LIN {X 0,Y 401.03,Z 373.683,A -85,B 0,C 180,E1 -11453.633,E2 -11453.633} C_VEL
LIN {X 0,Y 401.846,Z 358.726,A -85,B 0,C 180,E1 -11454.448,E2 -11454.448} C_VEL
LIN {X 0,Y 397.42,Z 344.712,A -85,B 0,C 180,E1 -11455.362,E2 -11455.362} C_VEL
LIN {X 0,Y 391.491,Z 329.461,A -85,B 0,C 180,E1 -11456.225,E2 -11456.225} C_VEL
LIN {X 0,Y 390.297,Z 326.311,A -85,B 0,C 180,E1 -11456.415,E2 -11456.415} C_VEL
LIN {X 0,Y 390.293,Z 322.173,A -85,B 0,C 180,E1 -11459.09,E2 -11459.09} C_VEL
LIN {X 0,Y 390.321,Z 317.773,A -85,B 0,C 180,E1 -11462.192,E2 -11462.192} C_VEL
LIN {X 0,Y 390.35,Z 313.687,A -85,B 0,C 180,E1 -11465.179,E2 -11465.179} C_VEL
LIN {X 0,Y 390.43,Z 310.287,A -85,B 0,C 180,E1 -11467.736,E2 -11467.736} C_VEL
LIN {X 0,Y 390.446,Z 306.037,A -85,B 0,C 180,E1 -11470.887,E2 -11470.887} C_VEL
LIN {X 0,Y 390.052,Z 302.527,A -85,B 0,C 180,E1 -11473.545,E2 -11473.545} C_VEL
LIN {X 0,Y 390.057,Z 302.527,A -85,B 0,C 180,E1 -11476.789,E2 -11476.789} C_VEL
LIN {X 0,Y 390.056,Z 302.524,A -85,B 0,C 180,E1 -11479.56,E2 -11479.56} C_VEL
LIN {X 0,Y 390.042,Z 302.525,A -85,B 0,C 180,E1 -11482.449,E2 -11482.449} C_VEL
LIN {X 0,Y 390.068,Z 302.518,A -85,B 0,C 180,E1 -11485.975,E2 -11485.975} C_VEL
LIN {X 0,Y 390.036,Z 302.519,A -85,B 0,C 180,E1 -11489.7,E2 -11489.7} C_VEL
LIN {X 0,Y 390.033,Z 302.52,A -85,B 0,C 180,E1 -11493.226,E2 -11493.226} C_VEL
LIN {X 0,Y 390.069,Z 302.521,A -85,B 0,C 180,E1 -11496.763,E2 -11496.763} C_VEL
LIN {X 0,Y 390.103,Z 302.515,A -85,B 0,C 180,E1 -11499.983,E2 -11499.983} C_VEL
LIN {X 0,Y 390.138,Z 302.5,A -85,B 0,C 180,E1 -11503.248,E2 -11503.248} C_VEL
LIN {X 0,Y 390.195,Z 302.506,A -85,B 0,C 180,E1 -11506.561,E2 -11506.561} C_VEL
LIN {X 0,Y 390.167,Z 302.502,A -85,B 0,C 180,E1 -11509.623,E2 -11509.623} C_VEL
LIN {X 0,Y 390.247,Z 302.493,A -85,B 0,C 180,E1 -11512.758,E2 -11512.758} C_VEL
LIN {X 0,Y 390.211,Z 302.492,A -85,B 0,C 180,E1 -11514.833,E2 -11514.833} C_VEL
LIN {X 0,Y 390.418,Z 302.476,A -85,B 0,C 180,E1 -11517.937,E2 -11517.937} C_VEL
LIN {X 0,Y 390.549,Z 302.445,A -85,B 0,C 180,E1 -11520,E2 -11520} C_VEL
LIN {X 0,Y 390.273,Z 302.496,A -85,B 0,C 180,E1 -11523.097,E2 -11523.097} C_VEL
LIN {X 0,Y 390.301,Z 302.482,A -85,B 0,C 180,E1 -11526.202,E2 -11526.202} C_VEL
LIN {X 0,Y 390.194,Z 302.502,A -85,B 0,C 180,E1 -11529.329,E2 -11529.329} C_VEL
LIN {X 0,Y 390.171,Z 302.506,A -85,B 0,C 180,E1 -11532.483,E2 -11532.483} C_VEL
LIN {X 0,Y 390.138,Z 302.501,A -85,B 0,C 180,E1 -11535.677,E2 -11535.677} C_VEL
LIN {X 0,Y 390.102,Z 302.519,A -85,B 0,C 180,E1 -11538.922,E2 -11538.922} C_VEL
LIN {X 0,Y 390.036,Z 302.515,A -85,B 0,C 180,E1 -11542.234,E2 -11542.234} C_VEL
LIN {X 0,Y 390.049,Z 302.516,A -85,B 0,C 180,E1 -11545.722,E2 -11545.722} C_VEL
LIN {X 0,Y 390.032,Z 302.526,A -85,B 0,C 180,E1 -11549.112,E2 -11549.112} C_VEL
LIN {X 0,Y 390.042,Z 302.524,A -85,B 0,C 180,E1 -11552.721,E2 -11552.721} C_VEL
LIN {X 0,Y 390.055,Z 302.523,A -85,B 0,C 180,E1 -11555.825,E2 -11555.825} C_VEL
LIN {X 0,Y 390.065,Z 302.523,A -85,B 0,C 180,E1 -11559.218,E2 -11559.218} C_VEL
LIN {X 0,Y 390.042,Z 302.546,A -85,B 0,C 180,E1 -11561.744,E2 -11561.744} C_VEL
LIN {X 0,Y 392.326,Z 311.892,A -85,B 0,C 180,E1 -11565.039,E2 -11565.039} C_VEL
LIN {X 0,Y 395.159,Z 323.516,A -85,B 0,C 180,E1 -11568.849,E2 -11568.849} C_VEL
LIN {X 0,Y 398.138,Z 335.816,A -85,B 0,C 180,E1 -11572.593,E2 -11572.593} C_VEL
LIN {X 0,Y 398.472,Z 338.892,A -85,B 0,C 180,E1 -11573.469,E2 -11573.469} C_VEL
LIN {X 0,Y 396.461,Z 351.383,A -85,B 0,C 180,E1 -11576.665,E2 -11576.665} C_VEL
LIN {X 0,Y 394.575,Z 365.042,A -85,B 0,C 180,E1 -11580.085,E2 -11580.085} C_VEL
LIN {X 0,Y 392.745,Z 380.859,A -85,B 0,C 180,E1 -11583.952,E2 -11583.952} C_VEL
LIN {X 0,Y 396.794,Z 403.736,A -85,B 0,C 180,E1 -11584.777,E2 -11584.777} C_VEL
LIN {X 0,Y 398.586,Z 417.426,A -85,B 0,C 180,E1 -11585.407,E2 -11585.407} C_VEL
LIN {X 0,Y 399.347,Z 429.472,A -85,B 0,C 180,E1 -11586.051,E2 -11586.051} C_VEL
LIN {X 0,Y 398.063,Z 444.07,A -85,B 0,C 180,E1 -11586.911,E2 -11586.911} C_VEL
LIN {X 0,Y 396.506,Z 458.695,A -85,B 0,C 180,E1 -11588.011,E2 -11588.011} C_VEL
LIN {X 0,Y 394.957,Z 472.268,A -85,B 0,C 180,E1 -11589.289,E2 -11589.289} C_VEL
LIN {X 0,Y 393.553,Z 484.615,A -85,B 0,C 180,E1 -11590.709,E2 -11590.709} C_VEL
LIN {X 0,Y 392.203,Z 495.885,A -85,B 0,C 180,E1 -11592.264,E2 -11592.264} C_VEL
LIN {X 0,Y 391.183,Z 505.396,A -85,B 0,C 180,E1 -11593.831,E2 -11593.831} C_VEL
LIN {X 0,Y 390.271,Z 514.747,A -85,B 0,C 180,E1 -11595.664,E2 -11595.664} C_VEL
LIN {X 0,Y 389.615,Z 522.521,A -85,B 0,C 180,E1 -11597.499,E2 -11597.499} C_VEL
LIN {X 0,Y 389.166,Z 529.796,A -85,B 0,C 180,E1 -11599.596,E2 -11599.596} C_VEL
LIN {X 0,Y 389.001,Z 535.531,A -85,B 0,C 180,E1 -11601.69,E2 -11601.69} C_VEL
LIN {X 0,Y 389.046,Z 539.872,A -85,B 0,C 180,E1 -11603.778,E2 -11603.778} C_VEL
LIN {X 0,Y 389.039,Z 542.91,A -85,B 0,C 180,E1 -11605.856,E2 -11605.856} C_VEL
LIN {X 0,Y 389.189,Z 544.737,A -85,B 0,C 180,E1 -11607.93,E2 -11607.93} C_VEL
LIN {X 0,Y 389.08,Z 545.347,A -85,B 0,C 180,E1 -11610,E2 -11610} C_VEL
LIN {X 0,Y 389.187,Z 544.737,A -85,B 0,C 180,E1 -11612.07,E2 -11612.07} C_VEL
LIN {X 0,Y 389.089,Z 542.914,A -85,B 0,C 180,E1 -11614.144,E2 -11614.144} C_VEL
LIN {X 0,Y 389.076,Z 539.867,A -85,B 0,C 180,E1 -11616.222,E2 -11616.222} C_VEL
LIN {X 0,Y 389.06,Z 535.519,A -85,B 0,C 180,E1 -11618.309,E2 -11618.309} C_VEL
LIN {X 0,Y 389.195,Z 529.78,A -85,B 0,C 180,E1 -11620.404,E2 -11620.404} C_VEL
LIN {X 0,Y 389.64,Z 522.506,A -85,B 0,C 180,E1 -11622.501,E2 -11622.501} C_VEL
LIN {X 0,Y 390.283,Z 514.721,A -85,B 0,C 180,E1 -11624.336,E2 -11624.336} C_VEL
LIN {X 0,Y 391.158,Z 505.355,A -85,B 0,C 180,E1 -11626.17,E2 -11626.17} C_VEL
LIN {X 0,Y 392.253,Z 495.847,A -85,B 0,C 180,E1 -11627.734,E2 -11627.734} C_VEL
LIN {X 0,Y 393.271,Z 486.53,A -85,B 0,C 180,E1 -11629.035,E2 -11629.035} C_VEL
LIN {X 0,Y 394.675,Z 474.561,A -85,B 0,C 180,E1 -11630.455,E2 -11630.455} C_VEL
LIN {X 0,Y 396.187,Z 461.487,A -85,B 0,C 180,E1 -11631.735,E2 -11631.735} C_VEL
LIN {X 0,Y 397.585,Z 448.807,A -85,B 0,C 180,E1 -11632.748,E2 -11632.748} C_VEL
LIN {X 0,Y 398.922,Z 434.386,A -85,B 0,C 180,E1 -11633.673,E2 -11633.673} C_VEL
LIN {X 0,Y 399.351,Z 427.194,A -85,B 0,C 180,E1 -11634.06,E2 -11634.06} C_VEL
LIN {X 0,Y 398.169,Z 411.419,A -85,B 0,C 180,E1 -11634.857,E2 -11634.857} C_VEL
LIN {X 0,Y 397.083,Z 401.601,A -85,B 0,C 180,E1 -11635.344,E2 -11635.344} C_VEL
LIN {X 0,Y 394.918,Z 387.953,A -85,B 0,C 180,E1 -11636.086,E2 -11636.086} C_VEL
LIN {X 0,Y 392.929,Z 378.662,A -85,B 0,C 180,E1 -11636.619,E2 -11636.619} C_VEL
LIN {X 0,Y 394.825,Z 365.115,A -85,B 0,C 180,E1 -11640.19,E2 -11640.19} C_VEL
LIN {X 0,Y 396.932,Z 354.413,A -85,B 0,C 180,E1 -11643.291,E2 -11643.291} C_VEL
LIN {X 0,Y 399.879,Z 343.943,A -85,B 0,C 180,E1 -11646.696,E2 -11646.696} C_VEL
LIN {X 0,Y 399.578,Z 340.879,A -85,B 0,C 180,E1 -11647.996,E2 -11647.996} C_VEL
LIN {X 0,Y 398.234,Z 335.574,A -85,B 0,C 180,E1 -11650.767,E2 -11650.767} C_VEL
LIN {X 0,Y 397.006,Z 331.283,A -85,B 0,C 180,E1 -11653.662,E2 -11653.662} C_VEL
LIN {X 0,Y 395.994,Z 328.116,A -85,B 0,C 180,E1 -11656.691,E2 -11656.691} C_VEL
LIN {X 0,Y 395.412,Z 326.545,A -85,B 0,C 180,E1 -11658.881,E2 -11658.881} C_VEL
LIN {X 0,Y 394.819,Z 325.339,A -85,B 0,C 180,E1 -11661.557,E2 -11661.557} C_VEL
LIN {X 0,Y 394.321,Z 324.865,A -85,B 0,C 180,E1 -11663.974,E2 -11663.974} C_VEL
LIN {X 0,Y 393.477,Z 325.038,A -85,B 0,C 180,E1 -11667.599,E2 -11667.599} C_VEL
LIN {X 0,Y 392.817,Z 325.946,A -85,B 0,C 180,E1 -11671.244,E2 -11671.244} C_VEL
LIN {X 0,Y 392.385,Z 327.254,A -85,B 0,C 180,E1 -11674.541,E2 -11674.541} C_VEL
LIN {X 0,Y 392.066,Z 328.943,A -85,B 0,C 180,E1 -11677.887,E2 -11677.887} C_VEL
LIN {X 0,Y 391.986,Z 329.43,A -85,B 0,C 180,E1 -11678.684,E2 -11678.684} C_VEL
LIN {X 0,Y 393.349,Z 332.348,A -85,B 0,C 180,E1 -11678.997,E2 -11678.997} C_VEL
LIN {X 0,Y 398.107,Z 342.204,A -85,B 0,C 180,E1 -11680.134,E2 -11680.134} C_VEL
LIN {X 0,Y 401.264,Z 350.393,A -85,B 0,C 180,E1 -11681.049,E2 -11681.049} C_VEL
LIN {X 0,Y 400.997,Z 355.665,A -85,B 0,C 180,E1 -11681.457,E2 -11681.457} C_VEL
LIN {X 0,Y 399.708,Z 367.932,A -85,B 0,C 180,E1 -11682.503,E2 -11682.503} C_VEL
LIN {X 0,Y 398.232,Z 379.64,A -85,B 0,C 180,E1 -11683.73,E2 -11683.73} C_VEL
LIN {X 0,Y 396.864,Z 390.351,A -85,B 0,C 180,E1 -11685.121,E2 -11685.121} C_VEL
LIN {X 0,Y 395.58,Z 399.819,A -85,B 0,C 180,E1 -11686.646,E2 -11686.646} C_VEL
LIN {X 0,Y 394.376,Z 407.68,A -85,B 0,C 180,E1 -11688.174,E2 -11688.174} C_VEL
LIN {X 0,Y 393.313,Z 414.086,A -85,B 0,C 180,E1 -11689.707,E2 -11689.707} C_VEL
LIN {X 0,Y 392.54,Z 419.208,A -85,B 0,C 180,E1 -11691.247,E2 -11691.247} C_VEL
LIN {X 0,Y 391.71,Z 423.284,A -85,B 0,C 180,E1 -11692.785,E2 -11692.785} C_VEL
LIN {X 0,Y 391.315,Z 425.442,A -85,B 0,C 180,E1 -11693.814,E2 -11693.814} C_VEL
LIN {X 0,Y 390.95,Z 428.372,A -85,B 0,C 180,E1 -11695.877,E2 -11695.877} C_VEL
LIN {X 0,Y 390.674,Z 429.276,A -85,B 0,C 180,E1 -11696.906,E2 -11696.906} C_VEL
LIN {X 0,Y 390.434,Z 429.786,A -85,B 0,C 180,E1 -11697.937,E2 -11697.937} C_VEL
LIN {X 0,Y 390.308,Z 429.858,A -85,B 0,C 180,E1 -11698.968,E2 -11698.968} C_VEL
LIN {X 0,Y 390.151,Z 428.837,A -85,B 0,C 180,E1 -11701.032,E2 -11701.032} C_VEL
LIN {X 0,Y 390.034,Z 427.759,A -85,B 0,C 180,E1 -11702.065,E2 -11702.065} C_VEL
LIN {X 0,Y 389.964,Z 426.237,A -85,B 0,C 180,E1 -11703.099,E2 -11703.099} C_VEL
LIN {X 0,Y 390.195,Z 423.138,A -85,B 0,C 180,E1 -11704.649,E2 -11704.649} C_VEL
LIN {X 0,Y 390.507,Z 419.028,A -85,B 0,C 180,E1 -11706.199,E2 -11706.199} C_VEL
LIN {X 0,Y 390.863,Z 412.829,A -85,B 0,C 180,E1 -11708.01,E2 -11708.01} C_VEL
LIN {X 0,Y 391.364,Z 404.933,A -85,B 0,C 180,E1 -11709.823,E2 -11709.823} C_VEL
LIN {X 0,Y 391.878,Z 396.479,A -85,B 0,C 180,E1 -11711.378,E2 -11711.378} C_VEL
LIN {X 0,Y 392.607,Z 386.139,A -85,B 0,C 180,E1 -11712.93,E2 -11712.93} C_VEL
LIN {X 0,Y 393.342,Z 375.598,A -85,B 0,C 180,E1 -11714.222,E2 -11714.222} C_VEL
LIN {X 0,Y 394.133,Z 362.595,A -85,B 0,C 180,E1 -11715.514,E2 -11715.514} C_VEL
LIN {X 0,Y 394.779,Z 351.319,A -85,B 0,C 180,E1 -11716.416,E2 -11716.416} C_VEL
LIN {X 0,Y 395.172,Z 338.606,A -85,B 0,C 180,E1 -11717.231,E2 -11717.231} C_VEL
LIN {X 0,Y 391.437,Z 324.013,A -85,B 0,C 180,E1 -11718.105,E2 -11718.105} C_VEL
LIN {X 0,Y 389.442,Z 316.377,A -85,B 0,C 180,E1 -11718.495,E2 -11718.495} C_VEL
LIN {X 0,Y 389.452,Z 313.434,A -85,B 0,C 180,E1 -11721.157,E2 -11721.157} C_VEL
LIN {X 0,Y 389.474,Z 309.821,A -85,B 0,C 180,E1 -11724.521,E2 -11724.521} C_VEL
LIN {X 0,Y 389.487,Z 306.163,A -85,B 0,C 180,E1 -11727.979,E2 -11727.979} C_VEL
LIN {X 0,Y 389.532,Z 303.708,A -85,B 0,C 180,E1 -11730.343,E2 -11730.343} C_VEL
LIN {X 0,Y 389.562,Z 302.588,A -85,B 0,C 180,E1 -11731.546,E2 -11731.546} C_VEL
LIN {X 0,Y 389.926,Z 302.541,A -85,B 0,C 180,E1 -11735.224,E2 -11735.224} C_VEL
LIN {X 0,Y 390.041,Z 302.524,A -85,B 0,C 180,E1 -11737.78,E2 -11737.78} C_VEL
LIN {X 0,Y 390.059,Z 302.52,A -85,B 0,C 180,E1 -11740.821,E2 -11740.821} C_VEL
LIN {X 0,Y 390.057,Z 302.519,A -85,B 0,C 180,E1 -11743.886,E2 -11743.886} C_VEL
LIN {X 0,Y 390.065,Z 302.573,A -85,B 0,C 180,E1 -11746.623,E2 -11746.623} C_VEL
LIN {X 0,Y 390.479,Z 305.87,A -85,B 0,C 180,E1 -11749.107,E2 -11749.107} C_VEL
LIN {X 0,Y 390.433,Z 310.221,A -85,B 0,C 180,E1 -11752.375,E2 -11752.375} C_VEL
LIN {X 0,Y 390.33,Z 315.186,A -85,B 0,C 180,E1 -11756.071,E2 -11756.071} C_VEL
LIN {X 0,Y 390.32,Z 320.392,A -85,B 0,C 180,E1 -11759.8,E2 -11759.8} C_VEL
LIN {X 0,Y 390.263,Z 325.586,A -85,B 0,C 180,E1 -11763.243,E2 -11763.243} C_VEL
LIN {X 0,Y 390.271,Z 326.34,A -85,B 0,C 180,E1 -11763.717,E2 -11763.717} C_VEL
LIN {X 0,Y 394.457,Z 336.878,A -85,B 0,C 180,E1 -11764.277,E2 -11764.277} C_VEL
LIN {X 0,Y 399.267,Z 350.24,A -85,B 0,C 180,E1 -11765.087,E2 -11765.087} C_VEL
LIN {X 0,Y 401.888,Z 359.314,A -85,B 0,C 180,E1 -11765.683,E2 -11765.683} C_VEL
LIN {X 0,Y 400.935,Z 374.28,A -85,B 0,C 180,E1 -11766.497,E2 -11766.497} C_VEL
LIN {X 0,Y 399.752,Z 388.734,A -85,B 0,C 180,E1 -11767.518,E2 -11767.518} C_VEL
LIN {X 0,Y 398.42,Z 401.781,A -85,B 0,C 180,E1 -11768.665,E2 -11768.665} C_VEL
LIN {X 0,Y 397.026,Z 413.662,A -85,B 0,C 180,E1 -11769.933,E2 -11769.933} C_VEL
LIN {X 0,Y 395.681,Z 424.75,A -85,B 0,C 180,E1 -11771.354,E2 -11771.354} C_VEL
LIN {X 0,Y 394.294,Z 434.875,A -85,B 0,C 180,E1 -11772.896,E2 -11772.896} C_VEL
LIN {X 0,Y 392.9,Z 444.714,A -85,B 0,C 180,E1 -11774.691,E2 -11774.691} C_VEL
LIN {X 0,Y 391.888,Z 452.947,A -85,B 0,C 180,E1 -11776.518,E2 -11776.518} C_VEL
LIN {X 0,Y 390.902,Z 460.609,A -85,B 0,C 180,E1 -11778.593,E2 -11778.593} C_VEL
LIN {X 0,Y 390.19,Z 466.693,A -85,B 0,C 180,E1 -11780.671,E2 -11780.671} C_VEL
LIN {X 0,Y 389.699,Z 471.393,A -85,B 0,C 180,E1 -11782.747,E2 -11782.747} C_VEL
LIN {X 0,Y 389.383,Z 474.836,A -85,B 0,C 180,E1 -11784.822,E2 -11784.822} C_VEL
LIN {X 0,Y 389.298,Z 477.097,A -85,B 0,C 180,E1 -11786.895,E2 -11786.895} C_VEL
LIN {X 0,Y 389.012,Z 478.268,A -85,B 0,C 180,E1 -11788.965,E2 -11788.965} C_VEL
LIN {X 0,Y 389.012,Z 478.282,A -85,B 0,C 180,E1 -11791.035,E2 -11791.035} C_VEL
LIN {X 0,Y 389.279,Z 477.166,A -85,B 0,C 180,E1 -11793.105,E2 -11793.105} C_VEL
LIN {X 0,Y 389.382,Z 474.962,A -85,B 0,C 180,E1 -11795.178,E2 -11795.178} C_VEL
LIN {X 0,Y 389.704,Z 471.482,A -85,B 0,C 180,E1 -11797.305,E2 -11797.305} C_VEL
LIN {X 0,Y 390.147,Z 466.955,A -85,B 0,C 180,E1 -11799.33,E2 -11799.33} C_VEL
LIN {X 0,Y 390.91,Z 460.581,A -85,B 0,C 180,E1 -11801.511,E2 -11801.511} C_VEL
LIN {X 0,Y 391.87,Z 453.34,A -85,B 0,C 180,E1 -11803.482,E2 -11803.482} C_VEL
LIN {X 0,Y 392.934,Z 444.959,A -85,B 0,C 180,E1 -11805.354,E2 -11805.354} C_VEL
LIN {X 0,Y 392.757,Z 441.59,A -85,B 0,C 180,E1 -11806.057,E2 -11806.057} C_VEL
LIN {X 0,Y 390.887,Z 435.993,A -85,B 0,C 180,E1 -11807.228,E2 -11807.228} C_VEL
LIN {X 0,Y 389.054,Z 430.043,A -85,B 0,C 180,E1 -11808.36,E2 -11808.36} C_VEL
LIN {X 0,Y 388.921,Z 425.982,A -85,B 0,C 180,E1 -11808.99,E2 -11808.99} C_VEL
LIN {X 0,Y 390.227,Z 414.843,A -85,B 0,C 180,E1 -11810.463,E2 -11810.463} C_VEL
LIN {X 0,Y 391.894,Z 402.013,A -85,B 0,C 180,E1 -11811.846,E2 -11811.846} C_VEL
LIN {X 0,Y 393.303,Z 388.866,A -85,B 0,C 180,E1 -11813.01,E2 -11813.01} C_VEL
LIN {X 0,Y 394.564,Z 374.255,A -85,B 0,C 180,E1 -11814.045,E2 -11814.045} C_VEL
LIN {X 0,Y 395.332,Z 360.445,A -85,B 0,C 180,E1 -11814.821,E2 -11814.821} C_VEL
LIN {X 0,Y 390.892,Z 346.436,A -85,B 0,C 180,E1 -11815.774,E2 -11815.774} C_VEL
LIN {X 0,Y 385.604,Z 332.648,A -85,B 0,C 180,E1 -11816.593,E2 -11816.593} C_VEL
LIN {X 0,Y 383.337,Z 326.923,A -85,B 0,C 180,E1 -11816.914,E2 -11816.914} C_VEL
LIN {X 0,Y 383.334,Z 322.682,A -85,B 0,C 180,E1 -11819.671,E2 -11819.671} C_VEL
LIN {X 0,Y 383.344,Z 317.471,A -85,B 0,C 180,E1 -11823.367,E2 -11823.367} C_VEL
LIN {X 0,Y 383.37,Z 313.6,A -85,B 0,C 180,E1 -11826.233,E2 -11826.233} C_VEL
LIN {X 0,Y 383.496,Z 309.036,A -85,B 0,C 180,E1 -11829.673,E2 -11829.673} C_VEL
LIN {X 0,Y 383.438,Z 306.884,A -85,B 0,C 180,E1 -11831.287,E2 -11831.287} C_VEL
LIN {X 0,Y 383,Z 303.406,A -85,B 0,C 180,E1 -11834.023,E2 -11834.023} C_VEL
LIN {X 0,Y 383.01,Z 303.404,A -85,B 0,C 180,E1 -11837.24,E2 -11837.24} C_VEL
LIN {X 0,Y 383.013,Z 303.398,A -85,B 0,C 180,E1 -11840.414,E2 -11840.414} C_VEL
LIN {X 0,Y 383.025,Z 303.397,A -85,B 0,C 180,E1 -11844.044,E2 -11844.044} C_VEL
LIN {X 0,Y 382.987,Z 303.404,A -85,B 0,C 180,E1 -11847.578,E2 -11847.578} C_VEL
LIN {X 0,Y 382.976,Z 303.398,A -85,B 0,C 180,E1 -11850.299,E2 -11850.299} C_VEL
LIN {X 0,Y 383.002,Z 303.392,A -85,B 0,C 180,E1 -11854.045,E2 -11854.045} C_VEL
LIN {X 0,Y 382.993,Z 303.396,A -85,B 0,C 180,E1 -11857.334,E2 -11857.334} C_VEL
LIN {X 0,Y 383.058,Z 303.395,A -85,B 0,C 180,E1 -11860.716,E2 -11860.716} C_VEL
LIN {X 0,Y 383.081,Z 303.383,A -85,B 0,C 180,E1 -11864.027,E2 -11864.027} C_VEL
LIN {X 0,Y 383.136,Z 303.376,A -85,B 0,C 180,E1 -11867.284,E2 -11867.284} C_VEL
LIN {X 0,Y 383.143,Z 303.385,A -85,B 0,C 180,E1 -11870.498,E2 -11870.498} C_VEL
LIN {X 0,Y 383.241,Z 303.356,A -85,B 0,C 180,E1 -11873.683,E2 -11873.683} C_VEL
LIN {X 0,Y 383.385,Z 303.352,A -85,B 0,C 180,E1 -11877.899,E2 -11877.899} C_VEL
LIN {X 0,Y 383.518,Z 303.321,A -85,B 0,C 180,E1 -11880,E2 -11880} C_VEL
LIN {X 0,Y 383.211,Z 303.376,A -85,B 0,C 180,E1 -11883.154,E2 -11883.154} C_VEL
LIN {X 0,Y 383.259,Z 303.359,A -85,B 0,C 180,E1 -11886.317,E2 -11886.317} C_VEL
LIN {X 0,Y 383.144,Z 303.38,A -85,B 0,C 180,E1 -11889.502,E2 -11889.502} C_VEL
LIN {X 0,Y 383.125,Z 303.388,A -85,B 0,C 180,E1 -11893.536,E2 -11893.536} C_VEL
LIN {X 0,Y 383.094,Z 303.382,A -85,B 0,C 180,E1 -11897.454,E2 -11897.454} C_VEL
LIN {X 0,Y 383.028,Z 303.39,A -85,B 0,C 180,E1 -11900.647,E2 -11900.647} C_VEL
LIN {X 0,Y 383.013,Z 303.403,A -85,B 0,C 180,E1 -11903.809,E2 -11903.809} C_VEL
LIN {X 0,Y 382.991,Z 303.394,A -85,B 0,C 180,E1 -11907.307,E2 -11907.307} C_VEL
LIN {X 0,Y 382.981,Z 303.404,A -85,B 0,C 180,E1 -11910.919,E2 -11910.919} C_VEL
LIN {X 0,Y 383.017,Z 303.399,A -85,B 0,C 180,E1 -11914.668,E2 -11914.668} C_VEL
LIN {X 0,Y 382.996,Z 303.404,A -85,B 0,C 180,E1 -11917.903,E2 -11917.903} C_VEL
LIN {X 0,Y 383.014,Z 303.55,A -85,B 0,C 180,E1 -11921.209,E2 -11921.209} C_VEL
LIN {X 0,Y 385.349,Z 313.104,A -85,B 0,C 180,E1 -11924.661,E2 -11924.661} C_VEL
LIN {X 0,Y 387.987,Z 324.048,A -85,B 0,C 180,E1 -11928.348,E2 -11928.348} C_VEL
LIN {X 0,Y 390.441,Z 334.196,A -85,B 0,C 180,E1 -11931.536,E2 -11931.536} C_VEL
LIN {X 0,Y 391.584,Z 339.187,A -85,B 0,C 180,E1 -11933.041,E2 -11933.041} C_VEL
LIN {X 0,Y 390.582,Z 345.973,A -85,B 0,C 180,E1 -11934.845,E2 -11934.845} C_VEL
LIN {X 0,Y 388.287,Z 360.674,A -85,B 0,C 180,E1 -11938.643,E2 -11938.643} C_VEL
LIN {X 0,Y 386.353,Z 375.405,A -85,B 0,C 180,E1 -11942.364,E2 -11942.364} C_VEL
LIN {X 0,Y 385.859,Z 379.755,A -85,B 0,C 180,E1 -11943.448,E2 -11943.448} C_VEL
LIN {X 0,Y 389.905,Z 402.276,A -85,B 0,C 180,E1 -11944.271,E2 -11944.271} C_VEL
LIN {X 0,Y 391.981,Z 417.492,A -85,B 0,C 180,E1 -11944.993,E2 -11944.993} C_VEL
LIN {X 0,Y 392.739,Z 430.161,A -85,B 0,C 180,E1 -11945.696,E2 -11945.696} C_VEL
LIN {X 0,Y 391.357,Z 444.834,A -85,B 0,C 180,E1 -11946.594,E2 -11946.594} C_VEL
LIN {X 0,Y 389.847,Z 458.096,A -85,B 0,C 180,E1 -11947.615,E2 -11947.615} C_VEL
LIN {X 0,Y 388.22,Z 471.662,A -85,B 0,C 180,E1 -11948.912,E2 -11948.912} C_VEL
LIN {X 0,Y 386.764,Z 484.007,A -85,B 0,C 180,E1 -11950.357,E2 -11950.357} C_VEL
LIN {X 0,Y 385.366,Z 495.276,A -85,B 0,C 180,E1 -11951.939,E2 -11951.939} C_VEL
LIN {X 0,Y 384.084,Z 506.223,A -85,B 0,C 180,E1 -11953.797,E2 -11953.797} C_VEL
LIN {X 0,Y 383.161,Z 515.344,A -85,B 0,C 180,E1 -11955.664,E2 -11955.664} C_VEL
LIN {X 0,Y 382.445,Z 523.89,A -85,B 0,C 180,E1 -11957.8,E2 -11957.8} C_VEL
LIN {X 0,Y 382.035,Z 530.763,A -85,B 0,C 180,E1 -11959.935,E2 -11959.935} C_VEL
LIN {X 0,Y 381.909,Z 536.152,A -85,B 0,C 180,E1 -11962.067,E2 -11962.067} C_VEL
LIN {X 0,Y 381.974,Z 539.261,A -85,B 0,C 180,E1 -11963.662,E2 -11963.662} C_VEL
LIN {X 0,Y 381.951,Z 542.3,A -85,B 0,C 180,E1 -11965.779,E2 -11965.779} C_VEL
LIN {X 0,Y 382.118,Z 544.129,A -85,B 0,C 180,E1 -11967.892,E2 -11967.892} C_VEL
LIN {X 0,Y 382.023,Z 544.74,A -85,B 0,C 180,E1 -11970,E2 -11970} C_VEL
LIN {X 0,Y 382.134,Z 544.13,A -85,B 0,C 180,E1 -11972.108,E2 -11972.108} C_VEL
LIN {X 0,Y 382,Z 542.303,A -85,B 0,C 180,E1 -11974.221,E2 -11974.221} C_VEL
LIN {X 0,Y 382.025,Z 538.84,A -85,B 0,C 180,E1 -11976.576,E2 -11976.576} C_VEL
LIN {X 0,Y 381.978,Z 534.903,A -85,B 0,C 180,E1 -11978.464,E2 -11978.464} C_VEL
LIN {X 0,Y 382.139,Z 529.163,A -85,B 0,C 180,E1 -11980.598,E2 -11980.598} C_VEL
LIN {X 0,Y 382.559,Z 521.883,A -85,B 0,C 180,E1 -11982.736,E2 -11982.736} C_VEL
LIN {X 0,Y 383.307,Z 514.103,A -85,B 0,C 180,E1 -11984.603,E2 -11984.603} C_VEL
LIN {X 0,Y 384.258,Z 504.739,A -85,B 0,C 180,E1 -11986.469,E2 -11986.469} C_VEL
LIN {X 0,Y 385.598,Z 494.074,A -85,B 0,C 180,E1 -11988.23,E2 -11988.23} C_VEL
LIN {X 0,Y 386.851,Z 482.901,A -85,B 0,C 180,E1 -11989.778,E2 -11989.778} C_VEL
LIN {X 0,Y 388.432,Z 470.334,A -85,B 0,C 180,E1 -11991.215,E2 -11991.215} C_VEL
LIN {X 0,Y 389.89,Z 458.008,A -85,B 0,C 180,E1 -11992.383,E2 -11992.383} C_VEL
LIN {X 0,Y 391.375,Z 444.736,A -85,B 0,C 180,E1 -11993.404,E2 -11993.404} C_VEL
LIN {X 0,Y 392.717,Z 429.998,A -85,B 0,C 180,E1 -11994.306,E2 -11994.306} C_VEL
LIN {X 0,Y 391.837,Z 413.945,A -85,B 0,C 180,E1 -11995.167,E2 -11995.167} C_VEL
LIN {X 0,Y 389.945,Z 395.637,A -85,B 0,C 180,E1 -11996.232,E2 -11996.232} C_VEL
LIN {X 0,Y 387.037,Z 381.169,A -85,B 0,C 180,E1 -11997.095,E2 -11997.095} C_VEL
LIN {X 0,Y 386.274,Z 377.616,A -85,B 0,C 180,E1 -11997.32,E2 -11997.32} C_VEL
LIN {X 0,Y 388.031,Z 366.053,A -85,B 0,C 180,E1 -12000.474,E2 -12000.474} C_VEL
LIN {X 0,Y 390.019,Z 356.428,A -85,B 0,C 180,E1 -12003.34,E2 -12003.34} C_VEL
LIN {X 0,Y 393.072,Z 346.004,A -85,B 0,C 180,E1 -12006.796,E2 -12006.796} C_VEL
LIN {X 0,Y 392.84,Z 343.029,A -85,B 0,C 180,E1 -12008.078,E2 -12008.078} C_VEL
LIN {X 0,Y 391.821,Z 338.889,A -85,B 0,C 180,E1 -12010.22,E2 -12010.22} C_VEL
LIN {X 0,Y 390.534,Z 334.384,A -85,B 0,C 180,E1 -12013.145,E2 -12013.145} C_VEL
LIN {X 0,Y 389.475,Z 330.904,A -85,B 0,C 180,E1 -12016.203,E2 -12016.203} C_VEL
LIN {X 0,Y 388.553,Z 328.548,A -85,B 0,C 180,E1 -12019.437,E2 -12019.437} C_VEL
LIN {X 0,Y 387.989,Z 327.465,A -85,B 0,C 180,E1 -12021.985,E2 -12021.985} C_VEL
LIN {X 0,Y 387.349,Z 326.994,A -85,B 0,C 180,E1 -12024.734,E2 -12024.734} C_VEL
LIN {X 0,Y 386.541,Z 327.185,A -85,B 0,C 180,E1 -12028.179,E2 -12028.179} C_VEL
LIN {X 0,Y 385.89,Z 328.066,A -85,B 0,C 180,E1 -12031.737,E2 -12031.737} C_VEL
LIN {X 0,Y 385.451,Z 329.412,A -85,B 0,C 180,E1 -12035.206,E2 -12035.206} C_VEL
LIN {X 0,Y 385.215,Z 330.769,A -85,B 0,C 180,E1 -12037.931,E2 -12037.931} C_VEL
LIN {X 0,Y 386.537,Z 333.683,A -85,B 0,C 180,E1 -12038.268,E2 -12038.268} C_VEL
LIN {X 0,Y 391.47,Z 343.418,A -85,B 0,C 180,E1 -12039.494,E2 -12039.494} C_VEL
LIN {X 0,Y 394.968,Z 352.4,A -85,B 0,C 180,E1 -12040.575,E2 -12040.575} C_VEL
LIN {X 0,Y 395.241,Z 354.192,A -85,B 0,C 180,E1 -12040.749,E2 -12040.749} C_VEL
LIN {X 0,Y 393.79,Z 367.17,A -85,B 0,C 180,E1 -12041.836,E2 -12041.836} C_VEL
LIN {X 0,Y 392.192,Z 379.079,A -85,B 0,C 180,E1 -12043.071,E2 -12043.071} C_VEL
LIN {X 0,Y 390.554,Z 390.888,A -85,B 0,C 180,E1 -12044.608,E2 -12044.608} C_VEL
LIN {X 0,Y 389.412,Z 399.021,A -85,B 0,C 180,E1 -12045.898,E2 -12045.898} C_VEL
LIN {X 0,Y 388.022,Z 407.182,A -85,B 0,C 180,E1 -12047.447,E2 -12047.447} C_VEL
LIN {X 0,Y 386.933,Z 413.815,A -85,B 0,C 180,E1 -12049.006,E2 -12049.006} C_VEL
LIN {X 0,Y 385.933,Z 419.254,A -85,B 0,C 180,E1 -12050.567,E2 -12050.567} C_VEL
LIN {X 0,Y 385.187,Z 423.538,A -85,B 0,C 180,E1 -12052.135,E2 -12052.135} C_VEL
LIN {X 0,Y 384.421,Z 426.83,A -85,B 0,C 180,E1 -12053.703,E2 -12053.703} C_VEL
LIN {X 0,Y 383.985,Z 429.651,A -85,B 0,C 180,E1 -12055.802,E2 -12055.802} C_VEL
LIN {X 0,Y 383.721,Z 430.508,A -85,B 0,C 180,E1 -12056.85,E2 -12056.85} C_VEL
LIN {X 0,Y 383.446,Z 430.955,A -85,B 0,C 180,E1 -12057.899,E2 -12057.899} C_VEL
LIN {X 0,Y 383.311,Z 430.979,A -85,B 0,C 180,E1 -12058.95,E2 -12058.95} C_VEL
LIN {X 0,Y 383.147,Z 430.625,A -85,B 0,C 180,E1 -12060,E2 -12060} C_VEL
LIN {X 0,Y 383.127,Z 429.863,A -85,B 0,C 180,E1 -12061.051,E2 -12061.051} C_VEL
LIN {X 0,Y 383.009,Z 428.719,A -85,B 0,C 180,E1 -12062.103,E2 -12062.103} C_VEL
LIN {X 0,Y 382.995,Z 426.2,A -85,B 0,C 180,E1 -12063.682,E2 -12063.682} C_VEL
LIN {X 0,Y 383.229,Z 422.687,A -85,B 0,C 180,E1 -12065.261,E2 -12065.261} C_VEL
LIN {X 0,Y 383.553,Z 418.133,A -85,B 0,C 180,E1 -12066.84,E2 -12066.84} C_VEL
LIN {X 0,Y 383.91,Z 412.445,A -85,B 0,C 180,E1 -12068.421,E2 -12068.421} C_VEL
LIN {X 0,Y 384.474,Z 404.105,A -85,B 0,C 180,E1 -12070.267,E2 -12070.267} C_VEL
LIN {X 0,Y 385.002,Z 395.271,A -85,B 0,C 180,E1 -12071.851,E2 -12071.851} C_VEL
LIN {X 0,Y 385.754,Z 385.395,A -85,B 0,C 180,E1 -12073.298,E2 -12073.298} C_VEL
LIN {X 0,Y 386.582,Z 373.271,A -85,B 0,C 180,E1 -12074.745,E2 -12074.745} C_VEL
LIN {X 0,Y 387.333,Z 361.121,A -85,B 0,C 180,E1 -12075.915,E2 -12075.915} C_VEL
LIN {X 0,Y 388.141,Z 347.663,A -85,B 0,C 180,E1 -12076.943,E2 -12076.943} C_VEL
LIN {X 0,Y 388.428,Z 341.443,A -85,B 0,C 180,E1 -12077.34,E2 -12077.34} C_VEL
LIN {X 0,Y 385.984,Z 330.752,A -85,B 0,C 180,E1 -12078.031,E2 -12078.031} C_VEL
LIN {X 0,Y 382.405,Z 316.954,A -85,B 0,C 180,E1 -12078.761,E2 -12078.761} C_VEL
LIN {X 0,Y 382.408,Z 313.871,A -85,B 0,C 180,E1 -12081.566,E2 -12081.566} C_VEL
LIN {X 0,Y 382.419,Z 310.18,A -85,B 0,C 180,E1 -12085.005,E2 -12085.005} C_VEL
LIN {X 0,Y 382.438,Z 306.47,A -85,B 0,C 180,E1 -12088.542,E2 -12088.542} C_VEL
LIN {X 0,Y 382.487,Z 303.96,A -85,B 0,C 180,E1 -12090.963,E2 -12090.963} C_VEL
LIN {X 0,Y 382.585,Z 303.456,A -85,B 0,C 180,E1 -12092.326,E2 -12092.326} C_VEL
LIN {X 0,Y 382.953,Z 303.407,A -85,B 0,C 180,E1 -12095.964,E2 -12095.964} C_VEL
LIN {X 0,Y 383.005,Z 303.402,A -85,B 0,C 180,E1 -12098.601,E2 -12098.601} C_VEL
LIN {X 0,Y 382.986,Z 303.399,A -85,B 0,C 180,E1 -12101.347,E2 -12101.347} C_VEL
LIN {X 0,Y 382.997,Z 303.399,A -85,B 0,C 180,E1 -12104.303,E2 -12104.303} C_VEL
LIN {X 0,Y 383.042,Z 303.611,A -85,B 0,C 180,E1 -12106.35,E2 -12106.35} C_VEL
LIN {X 0,Y 383.463,Z 306.709,A -85,B 0,C 180,E1 -12108.715,E2 -12108.715} C_VEL
LIN {X 0,Y 383.473,Z 310.32,A -85,B 0,C 180,E1 -12111.455,E2 -12111.455} C_VEL
LIN {X 0,Y 383.405,Z 313.835,A -85,B 0,C 180,E1 -12114.085,E2 -12114.085} C_VEL
LIN {X 0,Y 383.315,Z 318.486,A -85,B 0,C 180,E1 -12117.501,E2 -12117.501} C_VEL
LIN {X 0,Y 383.327,Z 322.523,A -85,B 0,C 180,E1 -12120.328,E2 -12120.328} C_VEL
LIN {X 0,Y 383.344,Z 327.084,A -85,B 0,C 180,E1 -12123.213,E2 -12123.213} C_VEL
LIN {X 0,Y 385.702,Z 332.936,A -85,B 0,C 180,E1 -12123.524,E2 -12123.524} C_VEL
LIN {X 0,Y 391.326,Z 347.568,A -85,B 0,C 180,E1 -12124.406,E2 -12124.406} C_VEL
LIN {X 0,Y 395.212,Z 359.872,A -85,B 0,C 180,E1 -12125.243,E2 -12125.243} C_VEL
LIN {X 0,Y 395.297,Z 363.044,A -85,B 0,C 180,E1 -12125.422,E2 -12125.422} C_VEL
LIN {X 0,Y 394.284,Z 376.828,A -85,B 0,C 180,E1 -12126.216,E2 -12126.216} C_VEL
LIN {X 0,Y 393.221,Z 389.331,A -85,B 0,C 180,E1 -12127.124,E2 -12127.124} C_VEL
LIN {X 0,Y 391.856,Z 402.379,A -85,B 0,C 180,E1 -12128.289,E2 -12128.289} C_VEL
LIN {X 0,Y 390.371,Z 414.489,A -85,B 0,C 180,E1 -12129.603,E2 -12129.603} C_VEL
LIN {X 0,Y 388.99,Z 425.353,A -85,B 0,C 180,E1 -12131.021,E2 -12131.021} C_VEL
LIN {X 0,Y 387.534,Z 435.481,A -85,B 0,C 180,E1 -12132.588,E2 -12132.588} C_VEL
LIN {X 0,Y 386.276,Z 444.059,A -85,B 0,C 180,E1 -12134.162,E2 -12134.162} C_VEL
LIN {X 0,Y 385.158,Z 452.476,A -85,B 0,C 180,E1 -12136.008,E2 -12136.008} C_VEL
LIN {X 0,Y 384.21,Z 459.471,A -85,B 0,C 180,E1 -12137.856,E2 -12137.856} C_VEL
LIN {X 0,Y 383.376,Z 465.931,A -85,B 0,C 180,E1 -12139.97,E2 -12139.97} C_VEL
LIN {X 0,Y 382.78,Z 470.978,A -85,B 0,C 180,E1 -12142.085,E2 -12142.085} C_VEL
LIN {X 0,Y 382.379,Z 473.884,A -85,B 0,C 180,E1 -12143.668,E2 -12143.668} C_VEL
LIN {X 0,Y 382.267,Z 476.718,A -85,B 0,C 180,E1 -12145.782,E2 -12145.782} C_VEL
LIN {X 0,Y 382.097,Z 478.427,A -85,B 0,C 180,E1 -12147.892,E2 -12147.892} C_VEL
LIN {X 0,Y 381.922,Z 479.03,A -85,B 0,C 180,E1 -12150,E2 -12150} C_VEL
LIN {X 0,Y 382.096,Z 478.467,A -85,B 0,C 180,E1 -12152.108,E2 -12152.108} C_VEL
LIN {X 0,Y 382.262,Z 476.813,A -85,B 0,C 180,E1 -12154.217,E2 -12154.217} C_VEL
LIN {X 0,Y 382.38,Z 474.04,A -85,B 0,C 180,E1 -12156.331,E2 -12156.331} C_VEL
LIN {X 0,Y 382.889,Z 470.042,A -85,B 0,C 180,E1 -12158.444,E2 -12158.444} C_VEL
LIN {X 0,Y 383.499,Z 464.733,A -85,B 0,C 180,E1 -12160.559,E2 -12160.559} C_VEL
LIN {X 0,Y 384.401,Z 457.952,A -85,B 0,C 180,E1 -12162.673,E2 -12162.673} C_VEL
LIN {X 0,Y 385.393,Z 450.701,A -85,B 0,C 180,E1 -12164.517,E2 -12164.517} C_VEL
LIN {X 0,Y 386.637,Z 441.901,A -85,B 0,C 180,E1 -12166.364,E2 -12166.364} C_VEL
LIN {X 0,Y 388.181,Z 431.265,A -85,B 0,C 180,E1 -12168.198,E2 -12168.198} C_VEL
LIN {X 0,Y 388.921,Z 425.982,A -85,B 0,C 180,E1 -12168.99,E2 -12168.99} C_VEL
LIN {X 0,Y 388.78,Z 421.875,A -85,B 0,C 180,E1 -12169.603,E2 -12169.603} C_VEL
LIN {X 0,Y 386.984,Z 415.144,A -85,B 0,C 180,E1 -12170.641,E2 -12170.641} C_VEL
LIN {X 0,Y 385.264,Z 408.011,A -85,B 0,C 180,E1 -12171.635,E2 -12171.635} C_VEL
LIN {X 0,Y 385.242,Z 403.284,A -85,B 0,C 180,E1 -12172.169,E2 -12172.169} C_VEL
LIN {X 0,Y 386.81,Z 389.449,A -85,B 0,C 180,E1 -12173.419,E2 -12173.419} C_VEL
LIN {X 0,Y 388.123,Z 374.827,A -85,B 0,C 180,E1 -12174.47,E2 -12174.47} C_VEL
LIN {X 0,Y 388.919,Z 362.911,A -85,B 0,C 180,E1 -12175.152,E2 -12175.152} C_VEL
LIN {X 0,Y 385.625,Z 351.651,A -85,B 0,C 180,E1 -12175.952,E2 -12175.952} C_VEL
LIN {X 0,Y 380.639,Z 338.066,A -85,B 0,C 180,E1 -12176.832,E2 -12176.832} C_VEL
LIN {X 0,Y 376.483,Z 328.03,A -85,B 0,C 180,E1 -12177.411,E2 -12177.411} C_VEL
LIN {X 0,Y 376.376,Z 327.483,A -85,B 0,C 180,E1 -12177.464,E2 -12177.464} C_VEL
LIN {X 0,Y 376.374,Z 322.442,A -85,B 0,C 180,E1 -12180.8,E2 -12180.8} C_VEL
LIN {X 0,Y 376.414,Z 316.907,A -85,B 0,C 180,E1 -12184.762,E2 -12184.762} C_VEL
LIN {X 0,Y 376.502,Z 312.129,A -85,B 0,C 180,E1 -12188.372,E2 -12188.372} C_VEL
LIN {X 0,Y 376.485,Z 308.948,A -85,B 0,C 180,E1 -12190.795,E2 -12190.795} C_VEL
LIN {X 0,Y 376.114,Z 305.088,A -85,B 0,C 180,E1 -12193.739,E2 -12193.739} C_VEL
LIN {X 0,Y 375.946,Z 304.285,A -85,B 0,C 180,E1 -12194.48,E2 -12194.48} C_VEL
LIN {X 0,Y 375.932,Z 304.285,A -85,B 0,C 180,E1 -12197.7,E2 -12197.7} C_VEL
LIN {X 0,Y 375.96,Z 304.276,A -85,B 0,C 180,E1 -12200.537,E2 -12200.537} C_VEL
LIN {X 0,Y 375.963,Z 304.274,A -85,B 0,C 180,E1 -12203.495,E2 -12203.495} C_VEL
LIN {X 0,Y 375.96,Z 304.276,A -85,B 0,C 180,E1 -12205.888,E2 -12205.888} C_VEL
LIN {X 0,Y 375.961,Z 304.271,A -85,B 0,C 180,E1 -12209.687,E2 -12209.687} C_VEL
LIN {X 0,Y 375.918,Z 304.285,A -85,B 0,C 180,E1 -12212.135,E2 -12212.135} C_VEL
LIN {X 0,Y 375.973,Z 304.278,A -85,B 0,C 180,E1 -12215.717,E2 -12215.717} C_VEL
LIN {X 0,Y 375.998,Z 304.268,A -85,B 0,C 180,E1 -12219.198,E2 -12219.198} C_VEL
LIN {X 0,Y 376.032,Z 304.258,A -85,B 0,C 180,E1 -12222.6,E2 -12222.6} C_VEL
LIN {X 0,Y 376.09,Z 304.263,A -85,B 0,C 180,E1 -12226.342,E2 -12226.342} C_VEL
LIN {X 0,Y 376.113,Z 304.258,A -85,B 0,C 180,E1 -12230.318,E2 -12230.318} C_VEL
LIN {X 0,Y 376.2,Z 304.233,A -85,B 0,C 180,E1 -12233.564,E2 -12233.564} C_VEL
LIN {X 0,Y 376.351,Z 304.228,A -85,B 0,C 180,E1 -12237.859,E2 -12237.859} C_VEL
LIN {X 0,Y 376.487,Z 304.196,A -85,B 0,C 180,E1 -12240,E2 -12240} C_VEL
LIN {X 0,Y 376.344,Z 304.233,A -85,B 0,C 180,E1 -12242.14,E2 -12242.14} C_VEL
LIN {X 0,Y 376.217,Z 304.237,A -85,B 0,C 180,E1 -12246.435,E2 -12246.435} C_VEL
LIN {X 0,Y 376.114,Z 304.253,A -85,B 0,C 180,E1 -12249.681,E2 -12249.681} C_VEL
LIN {X 0,Y 376.089,Z 304.266,A -85,B 0,C 180,E1 -12253.658,E2 -12253.658} C_VEL
LIN {X 0,Y 376.042,Z 304.262,A -85,B 0,C 180,E1 -12257.607,E2 -12257.607} C_VEL
LIN {X 0,Y 375.978,Z 304.267,A -85,B 0,C 180,E1 -12260.832,E2 -12260.832} C_VEL
LIN {X 0,Y 375.971,Z 304.278,A -85,B 0,C 180,E1 -12264.283,E2 -12264.283} C_VEL
LIN {X 0,Y 375.933,Z 304.278,A -85,B 0,C 180,E1 -12267.864,E2 -12267.864} C_VEL
LIN {X 0,Y 375.957,Z 304.28,A -85,B 0,C 180,E1 -12271.562,E2 -12271.562} C_VEL
LIN {X 0,Y 375.956,Z 304.281,A -85,B 0,C 180,E1 -12275.416,E2 -12275.416} C_VEL
LIN {X 0,Y 375.97,Z 304.28,A -85,B 0,C 180,E1 -12278.27,E2 -12278.27} C_VEL
LIN {X 0,Y 376.002,Z 304.404,A -85,B 0,C 180,E1 -12280.611,E2 -12280.611} C_VEL
LIN {X 0,Y 378.258,Z 313.981,A -85,B 0,C 180,E1 -12284.166,E2 -12284.166} C_VEL
LIN {X 0,Y 380.652,Z 323.918,A -85,B 0,C 180,E1 -12287.606,E2 -12287.606} C_VEL
LIN {X 0,Y 383.174,Z 334.244,A -85,B 0,C 180,E1 -12290.959,E2 -12290.959} C_VEL
LIN {X 0,Y 384.637,Z 340.602,A -85,B 0,C 180,E1 -12292.917,E2 -12292.917} C_VEL
LIN {X 0,Y 383.815,Z 346.228,A -85,B 0,C 180,E1 -12294.453,E2 -12294.453} C_VEL
LIN {X 0,Y 381.665,Z 359.183,A -85,B 0,C 180,E1 -12297.892,E2 -12297.892} C_VEL
LIN {X 0,Y 379.7,Z 373.226,A -85,B 0,C 180,E1 -12301.536,E2 -12301.536} C_VEL
LIN {X 0,Y 379.018,Z 378.638,A -85,B 0,C 180,E1 -12302.928,E2 -12302.928} C_VEL
LIN {X 0,Y 382.989,Z 400.209,A -85,B 0,C 180,E1 -12303.723,E2 -12303.723} C_VEL
LIN {X 0,Y 385.161,Z 415.871,A -85,B 0,C 180,E1 -12304.471,E2 -12304.471} C_VEL
LIN {X 0,Y 386.156,Z 429.575,A -85,B 0,C 180,E1 -12305.254,E2 -12305.254} C_VEL
LIN {X 0,Y 384.769,Z 444.563,A -85,B 0,C 180,E1 -12306.195,E2 -12306.195} C_VEL
LIN {X 0,Y 383.058,Z 458.939,A -85,B 0,C 180,E1 -12307.339,E2 -12307.339} C_VEL
LIN {X 0,Y 381.357,Z 472.242,A -85,B 0,C 180,E1 -12308.656,E2 -12308.656} C_VEL
LIN {X 0,Y 379.993,Z 483.399,A -85,B 0,C 180,E1 -12309.992,E2 -12309.992} C_VEL
LIN {X 0,Y 378.545,Z 494.666,A -85,B 0,C 180,E1 -12311.602,E2 -12311.602} C_VEL
LIN {X 0,Y 377.183,Z 505.611,A -85,B 0,C 180,E1 -12313.492,E2 -12313.492} C_VEL
LIN {X 0,Y 376.197,Z 514.73,A -85,B 0,C 180,E1 -12315.392,E2 -12315.392} C_VEL
LIN {X 0,Y 375.404,Z 523.273,A -85,B 0,C 180,E1 -12317.567,E2 -12317.567} C_VEL
LIN {X 0,Y 374.963,Z 530.147,A -85,B 0,C 180,E1 -12319.743,E2 -12319.743} C_VEL
LIN {X 0,Y 374.832,Z 535.539,A -85,B 0,C 180,E1 -12321.916,E2 -12321.916} C_VEL
LIN {X 0,Y 374.903,Z 538.65,A -85,B 0,C 180,E1 -12323.542,E2 -12323.542} C_VEL
LIN {X 0,Y 374.864,Z 541.689,A -85,B 0,C 180,E1 -12325.699,E2 -12325.699} C_VEL
LIN {X 0,Y 375.035,Z 543.52,A -85,B 0,C 180,E1 -12327.852,E2 -12327.852} C_VEL
LIN {X 0,Y 374.967,Z 544.133,A -85,B 0,C 180,E1 -12330,E2 -12330} C_VEL
LIN {X 0,Y 375.065,Z 543.522,A -85,B 0,C 180,E1 -12332.148,E2 -12332.148} C_VEL
LIN {X 0,Y 374.912,Z 541.691,A -85,B 0,C 180,E1 -12334.3,E2 -12334.3} C_VEL
LIN {X 0,Y 374.952,Z 538.436,A -85,B 0,C 180,E1 -12336.579,E2 -12336.579} C_VEL
LIN {X 0,Y 374.907,Z 534.288,A -85,B 0,C 180,E1 -12338.625,E2 -12338.625} C_VEL
LIN {X 0,Y 375.097,Z 528.548,A -85,B 0,C 180,E1 -12340.799,E2 -12340.799} C_VEL
LIN {X 0,Y 375.529,Z 521.264,A -85,B 0,C 180,E1 -12342.978,E2 -12342.978} C_VEL
LIN {X 0,Y 376.32,Z 513.484,A -85,B 0,C 180,E1 -12344.88,E2 -12344.88} C_VEL
LIN {X 0,Y 377.351,Z 504.122,A -85,B 0,C 180,E1 -12346.779,E2 -12346.779} C_VEL
LIN {X 0,Y 378.615,Z 494.621,A -85,B 0,C 180,E1 -12348.395,E2 -12348.395} C_VEL
LIN {X 0,Y 379.951,Z 483.326,A -85,B 0,C 180,E1 -12350.011,E2 -12350.011} C_VEL
LIN {X 0,Y 381.59,Z 470.976,A -85,B 0,C 180,E1 -12351.473,E2 -12351.473} C_VEL
LIN {X 0,Y 383.297,Z 457.406,A -85,B 0,C 180,E1 -12352.789,E2 -12352.789} C_VEL
LIN {X 0,Y 384.952,Z 443.015,A -85,B 0,C 180,E1 -12353.906,E2 -12353.906} C_VEL
LIN {X 0,Y 386.145,Z 429.401,A -85,B 0,C 180,E1 -12354.747,E2 -12354.747} C_VEL
LIN {X 0,Y 385.395,Z 415.2,A -85,B 0,C 180,E1 -12355.567,E2 -12355.567} C_VEL
LIN {X 0,Y 384.079,Z 398.56,A -85,B 0,C 180,E1 -12356.652,E2 -12356.652} C_VEL
LIN {X 0,Y 381.972,Z 386.71,A -85,B 0,C 180,E1 -12357.407,E2 -12357.407} C_VEL
LIN {X 0,Y 379.631,Z 376.497,A -85,B 0,C 180,E1 -12358.088,E2 -12358.088} C_VEL
LIN {X 0,Y 381.44,Z 366.04,A -85,B 0,C 180,E1 -12361.058,E2 -12361.058} C_VEL
LIN {X 0,Y 384.086,Z 354.796,A -85,B 0,C 180,E1 -12364.573,E2 -12364.573} C_VEL
LIN {X 0,Y 386.243,Z 348.056,A -85,B 0,C 180,E1 -12366.903,E2 -12366.903} C_VEL
LIN {X 0,Y 386.327,Z 346.506,A -85,B 0,C 180,E1 -12367.548,E2 -12367.548} C_VEL
LIN {X 0,Y 385.235,Z 341.698,A -85,B 0,C 180,E1 -12369.984,E2 -12369.984} C_VEL
LIN {X 0,Y 383.934,Z 337.07,A -85,B 0,C 180,E1 -12372.928,E2 -12372.928} C_VEL
LIN {X 0,Y 382.907,Z 333.734,A -85,B 0,C 180,E1 -12375.776,E2 -12375.776} C_VEL
LIN {X 0,Y 382.075,Z 331.447,A -85,B 0,C 180,E1 -12378.533,E2 -12378.533} C_VEL
LIN {X 0,Y 381.436,Z 330.011,A -85,B 0,C 180,E1 -12381.211,E2 -12381.211} C_VEL
LIN {X 0,Y 380.725,Z 329.2,A -85,B 0,C 180,E1 -12384.314,E2 -12384.314} C_VEL
LIN {X 0,Y 379.881,Z 329.197,A -85,B 0,C 180,E1 -12387.553,E2 -12387.553} C_VEL
LIN {X 0,Y 379.166,Z 329.883,A -85,B 0,C 180,E1 -12391.189,E2 -12391.189} C_VEL
LIN {X 0,Y 378.665,Z 331.097,A -85,B 0,C 180,E1 -12394.73,E2 -12394.73} C_VEL
LIN {X 0,Y 378.407,Z 332.194,A -85,B 0,C 180,E1 -12397.11,E2 -12397.11} C_VEL
LIN {X 0,Y 379.8,Z 335.082,A -85,B 0,C 180,E1 -12397.49,E2 -12397.49} C_VEL
LIN {X 0,Y 384.595,Z 344.208,A -85,B 0,C 180,E1 -12398.744,E2 -12398.744} C_VEL
LIN {X 0,Y 388.756,Z 354.432,A -85,B 0,C 180,E1 -12400.063,E2 -12400.063} C_VEL
LIN {X 0,Y 389.215,Z 356.25,A -85,B 0,C 180,E1 -12400.276,E2 -12400.276} C_VEL
LIN {X 0,Y 387.664,Z 368.737,A -85,B 0,C 180,E1 -12401.366,E2 -12401.366} C_VEL
LIN {X 0,Y 385.927,Z 380.813,A -85,B 0,C 180,E1 -12402.651,E2 -12402.651} C_VEL
LIN {X 0,Y 384.332,Z 391.555,A -85,B 0,C 180,E1 -12404.08,E2 -12404.08} C_VEL
LIN {X 0,Y 382.811,Z 401.172,A -85,B 0,C 180,E1 -12405.65,E2 -12405.65} C_VEL
LIN {X 0,Y 381.348,Z 409.136,A -85,B 0,C 180,E1 -12407.223,E2 -12407.223} C_VEL
LIN {X 0,Y 380.177,Z 415.681,A -85,B 0,C 180,E1 -12408.825,E2 -12408.825} C_VEL
LIN {X 0,Y 379.141,Z 420.875,A -85,B 0,C 180,E1 -12410.397,E2 -12410.397} C_VEL
LIN {X 0,Y 378.338,Z 425.051,A -85,B 0,C 180,E1 -12411.992,E2 -12411.992} C_VEL
LIN {X 0,Y 377.52,Z 428.253,A -85,B 0,C 180,E1 -12413.587,E2 -12413.587} C_VEL
LIN {X 0,Y 377.043,Z 430.96,A -85,B 0,C 180,E1 -12415.724,E2 -12415.724} C_VEL
LIN {X 0,Y 376.761,Z 431.745,A -85,B 0,C 180,E1 -12416.792,E2 -12416.792} C_VEL
LIN {X 0,Y 376.455,Z 432.118,A -85,B 0,C 180,E1 -12417.86,E2 -12417.86} C_VEL
LIN {X 0,Y 376.311,Z 432.089,A -85,B 0,C 180,E1 -12418.93,E2 -12418.93} C_VEL
LIN {X 0,Y 376.128,Z 431.688,A -85,B 0,C 180,E1 -12420,E2 -12420} C_VEL
LIN {X 0,Y 376.103,Z 430.879,A -85,B 0,C 180,E1 -12421.071,E2 -12421.071} C_VEL
LIN {X 0,Y 375.984,Z 429.66,A -85,B 0,C 180,E1 -12422.143,E2 -12422.143} C_VEL
LIN {X 0,Y 375.961,Z 427.06,A -85,B 0,C 180,E1 -12423.751,E2 -12423.751} C_VEL
LIN {X 0,Y 376.219,Z 423.456,A -85,B 0,C 180,E1 -12425.36,E2 -12425.36} C_VEL
LIN {X 0,Y 376.615,Z 417.915,A -85,B 0,C 180,E1 -12427.233,E2 -12427.233} C_VEL
LIN {X 0,Y 377.107,Z 410.798,A -85,B 0,C 180,E1 -12429.114,E2 -12429.114} C_VEL
LIN {X 0,Y 377.617,Z 403.224,A -85,B 0,C 180,E1 -12430.726,E2 -12430.726} C_VEL
LIN {X 0,Y 378.176,Z 393.927,A -85,B 0,C 180,E1 -12432.34,E2 -12432.34} C_VEL
LIN {X 0,Y 379.06,Z 382.528,A -85,B 0,C 180,E1 -12433.947,E2 -12433.947} C_VEL
LIN {X 0,Y 379.872,Z 371.069,A -85,B 0,C 180,E1 -12435.251,E2 -12435.251} C_VEL
LIN {X 0,Y 380.648,Z 358.293,A -85,B 0,C 180,E1 -12436.438,E2 -12436.438} C_VEL
LIN {X 0,Y 381.439,Z 344.682,A -85,B 0,C 180,E1 -12437.423,E2 -12437.423} C_VEL
LIN {X 0,Y 381.495,Z 341.866,A -85,B 0,C 180,E1 -12437.606,E2 -12437.606} C_VEL
LIN {X 0,Y 378.004,Z 327.729,A -85,B 0,C 180,E1 -12438.519,E2 -12438.519} C_VEL
LIN {X 0,Y 375.376,Z 317.514,A -85,B 0,C 180,E1 -12439.053,E2 -12439.053} C_VEL
LIN {X 0,Y 375.35,Z 314.29,A -85,B 0,C 180,E1 -12441.992,E2 -12441.992} C_VEL
LIN {X 0,Y 375.398,Z 310.538,A -85,B 0,C 180,E1 -12445.505,E2 -12445.505} C_VEL
LIN {X 0,Y 375.406,Z 306.765,A -85,B 0,C 180,E1 -12449.127,E2 -12449.127} C_VEL
LIN {X 0,Y 375.455,Z 304.345,A -85,B 0,C 180,E1 -12451.609,E2 -12451.609} C_VEL
LIN {X 0,Y 375.844,Z 304.296,A -85,B 0,C 180,E1 -12455.428,E2 -12455.428} C_VEL
LIN {X 0,Y 375.974,Z 304.277,A -85,B 0,C 180,E1 -12458.27,E2 -12458.27} C_VEL
LIN {X 0,Y 375.937,Z 304.277,A -85,B 0,C 180,E1 -12461.601,E2 -12461.601} C_VEL
LIN {X 0,Y 375.924,Z 304.281,A -85,B 0,C 180,E1 -12465.269,E2 -12465.269} C_VEL
LIN {X 0,Y 375.968,Z 304.285,A -85,B 0,C 180,E1 -12465.765,E2 -12465.765} C_VEL
LIN {X 0,Y 376.418,Z 307.598,A -85,B 0,C 180,E1 -12468.317,E2 -12468.317} C_VEL
LIN {X 0,Y 376.528,Z 310.591,A -85,B 0,C 180,E1 -12470.608,E2 -12470.608} C_VEL
LIN {X 0,Y 376.443,Z 314.289,A -85,B 0,C 180,E1 -12473.397,E2 -12473.397} C_VEL
LIN {X 0,Y 376.395,Z 317.697,A -85,B 0,C 180,E1 -12475.933,E2 -12475.933} C_VEL
LIN {X 0,Y 376.371,Z 323.036,A -85,B 0,C 180,E1 -12479.723,E2 -12479.723} C_VEL
LIN {X 0,Y 376.335,Z 327.507,A -85,B 0,C 180,E1 -12482.662,E2 -12482.662} C_VEL
LIN {X 0,Y 382.856,Z 343.82,A -85,B 0,C 180,E1 -12483.631,E2 -12483.631} C_VEL
LIN {X 0,Y 387.524,Z 357.563,A -85,B 0,C 180,E1 -12484.568,E2 -12484.568} C_VEL
LIN {X 0,Y 388.947,Z 362.632,A -85,B 0,C 180,E1 -12484.936,E2 -12484.936} C_VEL
LIN {X 0,Y 388.014,Z 375.457,A -85,B 0,C 180,E1 -12485.665,E2 -12485.665} C_VEL
LIN {X 0,Y 386.731,Z 389.925,A -85,B 0,C 180,E1 -12486.718,E2 -12486.718} C_VEL
LIN {X 0,Y 385.302,Z 402.978,A -85,B 0,C 180,E1 -12487.901,E2 -12487.901} C_VEL
LIN {X 0,Y 383.871,Z 413.987,A -85,B 0,C 180,E1 -12489.105,E2 -12489.105} C_VEL
LIN {X 0,Y 382.53,Z 424.068,A -85,B 0,C 180,E1 -12490.409,E2 -12490.409} C_VEL
LIN {X 0,Y 381,Z 434.512,A -85,B 0,C 180,E1 -12492.002,E2 -12492.002} C_VEL
LIN {X 0,Y 379.477,Z 444.665,A -85,B 0,C 180,E1 -12493.871,E2 -12493.871} C_VEL
LIN {X 0,Y 378.286,Z 453.093,A -85,B 0,C 180,E1 -12495.751,E2 -12495.751} C_VEL
LIN {X 0,Y 377.285,Z 460.08,A -85,B 0,C 180,E1 -12497.63,E2 -12497.63} C_VEL
LIN {X 0,Y 376.388,Z 466.541,A -85,B 0,C 180,E1 -12499.782,E2 -12499.782} C_VEL
LIN {X 0,Y 375.769,Z 471.587,A -85,B 0,C 180,E1 -12501.936,E2 -12501.936} C_VEL
LIN {X 0,Y 375.354,Z 474.492,A -85,B 0,C 180,E1 -12503.549,E2 -12503.549} C_VEL
LIN {X 0,Y 375.221,Z 477.326,A -85,B 0,C 180,E1 -12505.703,E2 -12505.703} C_VEL
LIN {X 0,Y 375.055,Z 479.033,A -85,B 0,C 180,E1 -12507.852,E2 -12507.852} C_VEL
LIN {X 0,Y 374.872,Z 479.636,A -85,B 0,C 180,E1 -12510,E2 -12510} C_VEL
LIN {X 0,Y 375.053,Z 479.073,A -85,B 0,C 180,E1 -12512.148,E2 -12512.148} C_VEL
LIN {X 0,Y 375.216,Z 477.42,A -85,B 0,C 180,E1 -12514.297,E2 -12514.297} C_VEL
LIN {X 0,Y 375.354,Z 474.647,A -85,B 0,C 180,E1 -12516.45,E2 -12516.45} C_VEL
LIN {X 0,Y 375.874,Z 470.65,A -85,B 0,C 180,E1 -12518.602,E2 -12518.602} C_VEL
LIN {X 0,Y 376.538,Z 465.34,A -85,B 0,C 180,E1 -12520.757,E2 -12520.757} C_VEL
LIN {X 0,Y 377.482,Z 458.558,A -85,B 0,C 180,E1 -12522.91,E2 -12522.91} C_VEL
LIN {X 0,Y 378.404,Z 452.393,A -85,B 0,C 180,E1 -12524.521,E2 -12524.521} C_VEL
LIN {X 0,Y 379.627,Z 443.829,A -85,B 0,C 180,E1 -12526.399,E2 -12526.399} C_VEL
LIN {X 0,Y 380.949,Z 435.08,A -85,B 0,C 180,E1 -12528,E2 -12528} C_VEL
LIN {X 0,Y 382.428,Z 424.755,A -85,B 0,C 180,E1 -12529.596,E2 -12529.596} C_VEL
LIN {X 0,Y 383.915,Z 413.515,A -85,B 0,C 180,E1 -12531.053,E2 -12531.053} C_VEL
LIN {X 0,Y 385.242,Z 403.284,A -85,B 0,C 180,E1 -12532.169,E2 -12532.169} C_VEL
LIN {X 0,Y 385.189,Z 398.473,A -85,B 0,C 180,E1 -12532.683,E2 -12532.683} C_VEL
LIN {X 0,Y 381.88,Z 384.244,A -85,B 0,C 180,E1 -12534.222,E2 -12534.222} C_VEL
LIN {X 0,Y 381.427,Z 379.12,A -85,B 0,C 180,E1 -12534.656,E2 -12534.656} C_VEL
LIN {X 0,Y 381.535,Z 377.345,A -85,B 0,C 180,E1 -12534.782,E2 -12534.782} C_VEL
LIN {X 0,Y 382.42,Z 364.09,A -85,B 0,C 180,E1 -12535.574,E2 -12535.574} C_VEL
LIN {X 0,Y 378.172,Z 350.384,A -85,B 0,C 180,E1 -12536.585,E2 -12536.585} C_VEL
LIN {X 0,Y 372.777,Z 336.379,A -85,B 0,C 180,E1 -12537.509,E2 -12537.509} C_VEL
LIN {X 0,Y 369.407,Z 328.063,A -85,B 0,C 180,E1 -12538.027,E2 -12538.027} C_VEL
LIN {X 0,Y 369.421,Z 323.407,A -85,B 0,C 180,E1 -12541.119,E2 -12541.119} C_VEL
LIN {X 0,Y 369.457,Z 317.843,A -85,B 0,C 180,E1 -12545.118,E2 -12545.118} C_VEL
LIN {X 0,Y 369.531,Z 312.862,A -85,B 0,C 180,E1 -12548.874,E2 -12548.874} C_VEL
LIN {X 0,Y 369.468,Z 309.157,A -85,B 0,C 180,E1 -12551.741,E2 -12551.741} C_VEL
LIN {X 0,Y 368.929,Z 305.438,A -85,B 0,C 180,E1 -12554.6,E2 -12554.6} C_VEL
LIN {X 0,Y 368.877,Z 305.166,A -85,B 0,C 180,E1 -12555.175,E2 -12555.175} C_VEL
LIN {X 0,Y 368.883,Z 305.161,A -85,B 0,C 180,E1 -12558.177,E2 -12558.177} C_VEL
LIN {X 0,Y 368.906,Z 305.155,A -85,B 0,C 180,E1 -12561.36,E2 -12561.36} C_VEL
LIN {X 0,Y 368.937,Z 305.157,A -85,B 0,C 180,E1 -12565.146,E2 -12565.146} C_VEL
LIN {X 0,Y 368.929,Z 305.151,A -85,B 0,C 180,E1 -12569.046,E2 -12569.046} C_VEL
LIN {X 0,Y 368.858,Z 305.161,A -85,B 0,C 180,E1 -12572.788,E2 -12572.788} C_VEL
LIN {X 0,Y 368.926,Z 305.155,A -85,B 0,C 180,E1 -12576.119,E2 -12576.119} C_VEL
LIN {X 0,Y 368.936,Z 305.152,A -85,B 0,C 180,E1 -12579.947,E2 -12579.947} C_VEL
LIN {X 0,Y 368.968,Z 305.135,A -85,B 0,C 180,E1 -12583.398,E2 -12583.398} C_VEL
LIN {X 0,Y 369.058,Z 305.135,A -85,B 0,C 180,E1 -12586.79,E2 -12586.79} C_VEL
LIN {X 0,Y 369.063,Z 305.134,A -85,B 0,C 180,E1 -12590.132,E2 -12590.132} C_VEL
LIN {X 0,Y 369.16,Z 305.11,A -85,B 0,C 180,E1 -12593.441,E2 -12593.441} C_VEL
LIN {X 0,Y 369.316,Z 305.104,A -85,B 0,C 180,E1 -12597.819,E2 -12597.819} C_VEL
LIN {X 0,Y 369.457,Z 305.071,A -85,B 0,C 180,E1 -12600,E2 -12600} C_VEL
LIN {X 0,Y 369.308,Z 305.109,A -85,B 0,C 180,E1 -12602.181,E2 -12602.181} C_VEL
LIN {X 0,Y 369.178,Z 305.114,A -85,B 0,C 180,E1 -12606.559,E2 -12606.559} C_VEL
LIN {X 0,Y 369.064,Z 305.128,A -85,B 0,C 180,E1 -12609.868,E2 -12609.868} C_VEL
LIN {X 0,Y 369.037,Z 305.143,A -85,B 0,C 180,E1 -12613.772,E2 -12613.772} C_VEL
LIN {X 0,Y 369.001,Z 305.141,A -85,B 0,C 180,E1 -12617.768,E2 -12617.768} C_VEL
LIN {X 0,Y 368.909,Z 305.144,A -85,B 0,C 180,E1 -12621.221,E2 -12621.221} C_VEL
LIN {X 0,Y 368.925,Z 305.157,A -85,B 0,C 180,E1 -12624.778,E2 -12624.778} C_VEL
LIN {X 0,Y 368.915,Z 305.156,A -85,B 0,C 180,E1 -12628.441,E2 -12628.441} C_VEL
LIN {X 0,Y 368.909,Z 305.157,A -85,B 0,C 180,E1 -12630.987,E2 -12630.987} C_VEL
LIN {X 0,Y 368.935,Z 305.154,A -85,B 0,C 180,E1 -12634.853,E2 -12634.853} C_VEL
LIN {X 0,Y 368.905,Z 305.16,A -85,B 0,C 180,E1 -12638.64,E2 -12638.64} C_VEL
LIN {X 0,Y 368.971,Z 305.225,A -85,B 0,C 180,E1 -12640.005,E2 -12640.005} C_VEL
LIN {X 0,Y 371.098,Z 314.475,A -85,B 0,C 180,E1 -12643.526,E2 -12643.526} C_VEL
LIN {X 0,Y 373.58,Z 324.779,A -85,B 0,C 180,E1 -12647.197,E2 -12647.197} C_VEL
LIN {X 0,Y 376.002,Z 334.839,A -85,B 0,C 180,E1 -12650.543,E2 -12650.543} C_VEL
LIN {X 0,Y 377.608,Z 341.628,A -85,B 0,C 180,E1 -12652.69,E2 -12652.69} C_VEL
LIN {X 0,Y 377.493,Z 344.213,A -85,B 0,C 180,E1 -12653.433,E2 -12653.433} C_VEL
LIN {X 0,Y 375.276,Z 356.477,A -85,B 0,C 180,E1 -12656.785,E2 -12656.785} C_VEL
LIN {X 0,Y 373.051,Z 371.006,A -85,B 0,C 180,E1 -12660.671,E2 -12660.671} C_VEL
LIN {X 0,Y 372.187,Z 377.394,A -85,B 0,C 180,E1 -12662.354,E2 -12662.354} C_VEL
LIN {X 0,Y 376.463,Z 400.84,A -85,B 0,C 180,E1 -12663.27,E2 -12663.27} C_VEL
LIN {X 0,Y 378.664,Z 417.058,A -85,B 0,C 180,E1 -12664.085,E2 -12664.085} C_VEL
LIN {X 0,Y 379.546,Z 430.767,A -85,B 0,C 180,E1 -12664.908,E2 -12664.908} C_VEL
LIN {X 0,Y 378.074,Z 445.364,A -85,B 0,C 180,E1 -12665.861,E2 -12665.861} C_VEL
LIN {X 0,Y 376.46,Z 458.342,A -85,B 0,C 180,E1 -12666.919,E2 -12666.919} C_VEL
LIN {X 0,Y 374.696,Z 471.64,A -85,B 0,C 180,E1 -12668.257,E2 -12668.257} C_VEL
LIN {X 0,Y 373.197,Z 482.787,A -85,B 0,C 180,E1 -12669.611,E2 -12669.611} C_VEL
LIN {X 0,Y 371.73,Z 494.057,A -85,B 0,C 180,E1 -12671.252,E2 -12671.252} C_VEL
LIN {X 0,Y 370.284,Z 504.998,A -85,B 0,C 180,E1 -12673.175,E2 -12673.175} C_VEL
LIN {X 0,Y 369.225,Z 514.115,A -85,B 0,C 180,E1 -12675.11,E2 -12675.11} C_VEL
LIN {X 0,Y 368.361,Z 522.656,A -85,B 0,C 180,E1 -12677.326,E2 -12677.326} C_VEL
LIN {X 0,Y 367.911,Z 529.533,A -85,B 0,C 180,E1 -12679.545,E2 -12679.545} C_VEL
LIN {X 0,Y 367.744,Z 534.924,A -85,B 0,C 180,E1 -12681.759,E2 -12681.759} C_VEL
LIN {X 0,Y 367.843,Z 538.125,A -85,B 0,C 180,E1 -12683.469,E2 -12683.469} C_VEL
LIN {X 0,Y 367.78,Z 541.079,A -85,B 0,C 180,E1 -12685.616,E2 -12685.616} C_VEL
LIN {X 0,Y 367.956,Z 542.91,A -85,B 0,C 180,E1 -12687.811,E2 -12687.811} C_VEL
LIN {X 0,Y 367.914,Z 543.526,A -85,B 0,C 180,E1 -12690,E2 -12690} C_VEL
LIN {X 0,Y 367.983,Z 542.912,A -85,B 0,C 180,E1 -12692.189,E2 -12692.189} C_VEL
LIN {X 0,Y 367.827,Z 541.08,A -85,B 0,C 180,E1 -12694.383,E2 -12694.383} C_VEL
LIN {X 0,Y 367.88,Z 538.032,A -85,B 0,C 180,E1 -12696.582,E2 -12696.582} C_VEL
LIN {X 0,Y 367.813,Z 533.671,A -85,B 0,C 180,E1 -12698.793,E2 -12698.793} C_VEL
LIN {X 0,Y 368.054,Z 527.931,A -85,B 0,C 180,E1 -12701.009,E2 -12701.009} C_VEL
LIN {X 0,Y 368.528,Z 520.646,A -85,B 0,C 180,E1 -12703.229,E2 -12703.229} C_VEL
LIN {X 0,Y 369.337,Z 512.864,A -85,B 0,C 180,E1 -12705.168,E2 -12705.168} C_VEL
LIN {X 0,Y 370.469,Z 503.506,A -85,B 0,C 180,E1 -12707.1,E2 -12707.1} C_VEL
LIN {X 0,Y 371.953,Z 492.993,A -85,B 0,C 180,E1 -12708.901,E2 -12708.901} C_VEL
LIN {X 0,Y 373.243,Z 482.717,A -85,B 0,C 180,E1 -12710.387,E2 -12710.387} C_VEL
LIN {X 0,Y 374.927,Z 470.367,A -85,B 0,C 180,E1 -12711.874,E2 -12711.874} C_VEL
LIN {X 0,Y 376.717,Z 456.803,A -85,B 0,C 180,E1 -12713.211,E2 -12713.211} C_VEL
LIN {X 0,Y 378.457,Z 442.027,A -85,B 0,C 180,E1 -12714.372,E2 -12714.372} C_VEL
LIN {X 0,Y 379.52,Z 430.574,A -85,B 0,C 180,E1 -12715.095,E2 -12715.095} C_VEL
LIN {X 0,Y 379.209,Z 419.177,A -85,B 0,C 180,E1 -12715.832,E2 -12715.832} C_VEL
LIN {X 0,Y 378.33,Z 403.054,A -85,B 0,C 180,E1 -12716.97,E2 -12716.97} C_VEL
LIN {X 0,Y 376.498,Z 390.111,A -85,B 0,C 180,E1 -12717.859,E2 -12717.859} C_VEL
LIN {X 0,Y 373.14,Z 375.336,A -85,B 0,C 180,E1 -12718.923,E2 -12718.923} C_VEL
LIN {X 0,Y 375.614,Z 362.911,A -85,B 0,C 180,E1 -12722.65,E2 -12722.65} C_VEL
LIN {X 0,Y 378.865,Z 351.737,A -85,B 0,C 180,E1 -12726.414,E2 -12726.414} C_VEL
LIN {X 0,Y 379.524,Z 349.584,A -85,B 0,C 180,E1 -12727.225,E2 -12727.225} C_VEL
LIN {X 0,Y 379.333,Z 347.327,A -85,B 0,C 180,E1 -12728.256,E2 -12728.256} C_VEL
LIN {X 0,Y 378.021,Z 341.979,A -85,B 0,C 180,E1 -12731.225,E2 -12731.225} C_VEL
LIN {X 0,Y 376.971,Z 338.597,A -85,B 0,C 180,E1 -12733.615,E2 -12733.615} C_VEL
LIN {X 0,Y 375.896,Z 335.144,A -85,B 0,C 180,E1 -12736.817,E2 -12736.817} C_VEL
LIN {X 0,Y 374.937,Z 332.789,A -85,B 0,C 180,E1 -12740.222,E2 -12740.222} C_VEL
LIN {X 0,Y 374.259,Z 331.682,A -85,B 0,C 180,E1 -12743.065,E2 -12743.065} C_VEL
LIN {X 0,Y 373.517,Z 331.291,A -85,B 0,C 180,E1 -12745.883,E2 -12745.883} C_VEL
LIN {X 0,Y 372.683,Z 331.537,A -85,B 0,C 180,E1 -12749.392,E2 -12749.392} C_VEL
LIN {X 0,Y 372.069,Z 332.429,A -85,B 0,C 180,E1 -12753.042,E2 -12753.042} C_VEL
LIN {X 0,Y 371.651,Z 333.646,A -85,B 0,C 180,E1 -12756.214,E2 -12756.214} C_VEL
LIN {X 0,Y 374.267,Z 338.568,A -85,B 0,C 180,E1 -12756.945,E2 -12756.945} C_VEL
LIN {X 0,Y 379.154,Z 347.986,A -85,B 0,C 180,E1 -12758.348,E2 -12758.348} C_VEL
LIN {X 0,Y 383.093,Z 358.196,A -85,B 0,C 180,E1 -12759.756,E2 -12759.756} C_VEL
LIN {X 0,Y 381.566,Z 370.921,A -85,B 0,C 180,E1 -12760.917,E2 -12760.917} C_VEL
LIN {X 0,Y 379.722,Z 382.635,A -85,B 0,C 180,E1 -12762.219,E2 -12762.219} C_VEL
LIN {X 0,Y 377.847,Z 394.084,A -85,B 0,C 180,E1 -12763.8,E2 -12763.8} C_VEL
LIN {X 0,Y 376.263,Z 403.408,A -85,B 0,C 180,E1 -12765.395,E2 -12765.395} C_VEL
LIN {X 0,Y 374.708,Z 411.107,A -85,B 0,C 180,E1 -12766.993,E2 -12766.993} C_VEL
LIN {X 0,Y 373.448,Z 417.44,A -85,B 0,C 180,E1 -12768.603,E2 -12768.603} C_VEL
LIN {X 0,Y 372.361,Z 422.576,A -85,B 0,C 180,E1 -12770.22,E2 -12770.22} C_VEL
LIN {X 0,Y 371.482,Z 426.607,A -85,B 0,C 180,E1 -12771.843,E2 -12771.843} C_VEL
LIN {X 0,Y 370.609,Z 429.67,A -85,B 0,C 180,E1 -12773.467,E2 -12773.467} C_VEL
LIN {X 0,Y 370.095,Z 432.277,A -85,B 0,C 180,E1 -12775.644,E2 -12775.644} C_VEL
LIN {X 0,Y 369.797,Z 432.981,A -85,B 0,C 180,E1 -12776.732,E2 -12776.732} C_VEL
LIN {X 0,Y 369.484,Z 433.298,A -85,B 0,C 180,E1 -12777.82,E2 -12777.82} C_VEL
LIN {X 0,Y 369.33,Z 433.213,A -85,B 0,C 180,E1 -12778.91,E2 -12778.91} C_VEL
LIN {X 0,Y 369.11,Z 432.758,A -85,B 0,C 180,E1 -12780,E2 -12780} C_VEL
LIN {X 0,Y 369.079,Z 431.881,A -85,B 0,C 180,E1 -12781.091,E2 -12781.091} C_VEL
LIN {X 0,Y 368.958,Z 430.591,A -85,B 0,C 180,E1 -12782.183,E2 -12782.183} C_VEL
LIN {X 0,Y 368.929,Z 427.902,A -85,B 0,C 180,E1 -12783.823,E2 -12783.823} C_VEL
LIN {X 0,Y 369.209,Z 424.201,A -85,B 0,C 180,E1 -12785.462,E2 -12785.462} C_VEL
LIN {X 0,Y 369.587,Z 418.855,A -85,B 0,C 180,E1 -12787.279,E2 -12787.279} C_VEL
LIN {X 0,Y 370.002,Z 412.541,A -85,B 0,C 180,E1 -12788.988,E2 -12788.988} C_VEL
LIN {X 0,Y 370.542,Z 404.954,A -85,B 0,C 180,E1 -12790.657,E2 -12790.657} C_VEL
LIN {X 0,Y 371.102,Z 395.862,A -85,B 0,C 180,E1 -12792.302,E2 -12792.302} C_VEL
LIN {X 0,Y 372.036,Z 384.668,A -85,B 0,C 180,E1 -12793.937,E2 -12793.937} C_VEL
LIN {X 0,Y 372.844,Z 373.249,A -85,B 0,C 180,E1 -12795.301,E2 -12795.301} C_VEL
LIN {X 0,Y 373.638,Z 360.565,A -85,B 0,C 180,E1 -12796.529,E2 -12796.529} C_VEL
LIN {X 0,Y 374.499,Z 347.168,A -85,B 0,C 180,E1 -12797.556,E2 -12797.556} C_VEL
LIN {X 0,Y 374.449,Z 342.238,A -85,B 0,C 180,E1 -12797.888,E2 -12797.888} C_VEL
LIN {X 0,Y 370.637,Z 327.009,A -85,B 0,C 180,E1 -12798.876,E2 -12798.876} C_VEL
LIN {X 0,Y 368.305,Z 318.059,A -85,B 0,C 180,E1 -12799.363,E2 -12799.363} C_VEL
LIN {X 0,Y 368.321,Z 314.707,A -85,B 0,C 180,E1 -12802.434,E2 -12802.434} C_VEL
LIN {X 0,Y 368.349,Z 310.647,A -85,B 0,C 180,E1 -12806.266,E2 -12806.266} C_VEL
LIN {X 0,Y 368.374,Z 307.041,A -85,B 0,C 180,E1 -12809.738,E2 -12809.738} C_VEL
LIN {X 0,Y 368.4,Z 305.758,A -85,B 0,C 180,E1 -12811.003,E2 -12811.003} C_VEL
LIN {X 0,Y 368.545,Z 305.205,A -85,B 0,C 180,E1 -12812.958,E2 -12812.958} C_VEL
LIN {X 0,Y 368.857,Z 305.163,A -85,B 0,C 180,E1 -12816.204,E2 -12816.204} C_VEL
LIN {X 0,Y 368.904,Z 305.157,A -85,B 0,C 180,E1 -12818.953,E2 -12818.953} C_VEL
LIN {X 0,Y 368.884,Z 305.156,A -85,B 0,C 180,E1 -12822.009,E2 -12822.009} C_VEL
LIN {X 0,Y 368.931,Z 305.275,A -85,B 0,C 180,E1 -12825.4,E2 -12825.4} C_VEL
LIN {X 0,Y 369.471,Z 308.938,A -85,B 0,C 180,E1 -12828.259,E2 -12828.259} C_VEL
LIN {X 0,Y 369.551,Z 312.827,A -85,B 0,C 180,E1 -12831.235,E2 -12831.235} C_VEL
LIN {X 0,Y 369.475,Z 318.113,A -85,B 0,C 180,E1 -12835.204,E2 -12835.204} C_VEL
LIN {X 0,Y 369.398,Z 323.541,A -85,B 0,C 180,E1 -12839.09,E2 -12839.09} C_VEL
LIN {X 0,Y 369.389,Z 328.103,A -85,B 0,C 180,E1 -12842.104,E2 -12842.104} C_VEL
LIN {X 0,Y 371.533,Z 333.508,A -85,B 0,C 180,E1 -12842.413,E2 -12842.413} C_VEL
LIN {X 0,Y 376.98,Z 347.054,A -85,B 0,C 180,E1 -12843.283,E2 -12843.283} C_VEL
LIN {X 0,Y 381.493,Z 360.739,A -85,B 0,C 180,E1 -12844.27,E2 -12844.27} C_VEL
LIN {X 0,Y 382.47,Z 364.209,A -85,B 0,C 180,E1 -12844.54,E2 -12844.54} C_VEL
LIN {X 0,Y 381.39,Z 378.122,A -85,B 0,C 180,E1 -12845.368,E2 -12845.368} C_VEL
LIN {X 0,Y 380.239,Z 390.521,A -85,B 0,C 180,E1 -12846.296,E2 -12846.296} C_VEL
LIN {X 0,Y 378.747,Z 403.578,A -85,B 0,C 180,E1 -12847.498,E2 -12847.498} C_VEL
LIN {X 0,Y 377.242,Z 414.769,A -85,B 0,C 180,E1 -12848.743,E2 -12848.743} C_VEL
LIN {X 0,Y 375.872,Z 424.672,A -85,B 0,C 180,E1 -12850.048,E2 -12850.048} C_VEL
LIN {X 0,Y 374.264,Z 435.118,A -85,B 0,C 180,E1 -12851.667,E2 -12851.667} C_VEL
LIN {X 0,Y 372.675,Z 445.273,A -85,B 0,C 180,E1 -12853.568,E2 -12853.568} C_VEL
LIN {X 0,Y 371.415,Z 453.75,A -85,B 0,C 180,E1 -12855.495,E2 -12855.495} C_VEL
LIN {X 0,Y 370.367,Z 460.689,A -85,B 0,C 180,E1 -12857.395,E2 -12857.395} C_VEL
LIN {X 0,Y 369.416,Z 467.151,A -85,B 0,C 180,E1 -12859.587,E2 -12859.587} C_VEL
LIN {X 0,Y 368.758,Z 472.196,A -85,B 0,C 180,E1 -12861.782,E2 -12861.782} C_VEL
LIN {X 0,Y 368.332,Z 475.1,A -85,B 0,C 180,E1 -12863.426,E2 -12863.426} C_VEL
LIN {X 0,Y 368.175,Z 477.934,A -85,B 0,C 180,E1 -12865.621,E2 -12865.621} C_VEL
LIN {X 0,Y 368.014,Z 479.639,A -85,B 0,C 180,E1 -12867.811,E2 -12867.811} C_VEL
LIN {X 0,Y 367.824,Z 480.242,A -85,B 0,C 180,E1 -12870,E2 -12870} C_VEL
LIN {X 0,Y 368.011,Z 479.679,A -85,B 0,C 180,E1 -12872.189,E2 -12872.189} C_VEL
LIN {X 0,Y 368.171,Z 478.027,A -85,B 0,C 180,E1 -12874.379,E2 -12874.379} C_VEL
LIN {X 0,Y 368.331,Z 475.254,A -85,B 0,C 180,E1 -12876.574,E2 -12876.574} C_VEL
LIN {X 0,Y 368.878,Z 471.257,A -85,B 0,C 180,E1 -12878.767,E2 -12878.767} C_VEL
LIN {X 0,Y 369.588,Z 465.945,A -85,B 0,C 180,E1 -12880.962,E2 -12880.962} C_VEL
LIN {X 0,Y 370.572,Z 459.164,A -85,B 0,C 180,E1 -12883.155,E2 -12883.155} C_VEL
LIN {X 0,Y 371.668,Z 451.599,A -85,B 0,C 180,E1 -12885.14,E2 -12885.14} C_VEL
LIN {X 0,Y 373.083,Z 443.104,A -85,B 0,C 180,E1 -12886.977,E2 -12886.977} C_VEL
LIN {X 0,Y 374.759,Z 432.463,A -85,B 0,C 180,E1 -12888.874,E2 -12888.874} C_VEL
LIN {X 0,Y 376.271,Z 421.53,A -85,B 0,C 180,E1 -12890.5,E2 -12890.5} C_VEL
LIN {X 0,Y 377.998,Z 409.493,A -85,B 0,C 180,E1 -12891.973,E2 -12891.973} C_VEL
LIN {X 0,Y 379.614,Z 396.196,A -85,B 0,C 180,E1 -12893.311,E2 -12893.311} C_VEL
LIN {X 0,Y 381.033,Z 383.173,A -85,B 0,C 180,E1 -12894.374,E2 -12894.374} C_VEL
LIN {X 0,Y 381.535,Z 377.345,A -85,B 0,C 180,E1 -12894.782,E2 -12894.782} C_VEL
LIN {X 0,Y 381.489,Z 373.824,A -85,B 0,C 180,E1 -12895.042,E2 -12895.042} C_VEL
LIN {X 0,Y 380.157,Z 368.83,A -85,B 0,C 180,E1 -12895.478,E2 -12895.478} C_VEL
LIN {X 0,Y 377.904,Z 364.171,A -85,B 0,C 180,E1 -12895.934,E2 -12895.934} C_VEL
LIN {X 0,Y 372.724,Z 354.694,A -85,B 0,C 180,E1 -12896.837,E2 -12896.837} C_VEL
LIN {X 0,Y 371.402,Z 351.22,A -85,B 0,C 180,E1 -12897.098,E2 -12897.098} C_VEL
LIN {X 0,Y 366.07,Z 337.259,A -85,B 0,C 180,E1 -12898.047,E2 -12898.047} C_VEL
LIN {X 0,Y 362.499,Z 328.673,A -85,B 0,C 180,E1 -12898.598,E2 -12898.598} C_VEL
LIN {X 0,Y 362.457,Z 324.231,A -85,B 0,C 180,E1 -12901.569,E2 -12901.569} C_VEL
LIN {X 0,Y 362.499,Z 318.687,A -85,B 0,C 180,E1 -12905.565,E2 -12905.565} C_VEL
LIN {X 0,Y 362.561,Z 313.919,A -85,B 0,C 180,E1 -12909.161,E2 -12909.161} C_VEL
LIN {X 0,Y 362.534,Z 311.278,A -85,B 0,C 180,E1 -12911.232,E2 -12911.232} C_VEL
LIN {X 0,Y 362.144,Z 307.581,A -85,B 0,C 180,E1 -12914.106,E2 -12914.106} C_VEL
LIN {X 0,Y 361.819,Z 306.045,A -85,B 0,C 180,E1 -12915.465,E2 -12915.465} C_VEL
LIN {X 0,Y 361.827,Z 306.037,A -85,B 0,C 180,E1 -12918.669,E2 -12918.669} C_VEL
LIN {X 0,Y 361.866,Z 306.033,A -85,B 0,C 180,E1 -12921.575,E2 -12921.575} C_VEL
LIN {X 0,Y 361.874,Z 306.034,A -85,B 0,C 180,E1 -12924.655,E2 -12924.655} C_VEL
LIN {X 0,Y 361.838,Z 306.041,A -85,B 0,C 180,E1 -12928.37,E2 -12928.37} C_VEL
LIN {X 0,Y 361.865,Z 306.032,A -85,B 0,C 180,E1 -12930.952,E2 -12930.952} C_VEL
LIN {X 0,Y 361.882,Z 306.026,A -85,B 0,C 180,E1 -12934.706,E2 -12934.706} C_VEL
LIN {X 0,Y 361.861,Z 306.022,A -85,B 0,C 180,E1 -12938.345,E2 -12938.345} C_VEL
LIN {X 0,Y 361.92,Z 306.019,A -85,B 0,C 180,E1 -12942.085,E2 -12942.085} C_VEL
LIN {X 0,Y 361.962,Z 306.024,A -85,B 0,C 180,E1 -12945.38,E2 -12945.38} C_VEL
LIN {X 0,Y 361.971,Z 306.006,A -85,B 0,C 180,E1 -12948.804,E2 -12948.804} C_VEL
LIN {X 0,Y 362.078,Z 306.004,A -85,B 0,C 180,E1 -12952.191,E2 -12952.191} C_VEL
LIN {X 0,Y 362.096,Z 305.99,A -85,B 0,C 180,E1 -12954.431,E2 -12954.431} C_VEL
LIN {X 0,Y 362.28,Z 305.98,A -85,B 0,C 180,E1 -12957.776,E2 -12957.776} C_VEL
LIN {X 0,Y 362.427,Z 305.946,A -85,B 0,C 180,E1 -12960,E2 -12960} C_VEL
LIN {X 0,Y 362.271,Z 305.985,A -85,B 0,C 180,E1 -12962.223,E2 -12962.223} C_VEL
LIN {X 0,Y 362.14,Z 305.991,A -85,B 0,C 180,E1 -12966.687,E2 -12966.687} C_VEL
LIN {X 0,Y 362,Z 306.004,A -85,B 0,C 180,E1 -12970.063,E2 -12970.063} C_VEL
LIN {X 0,Y 361.998,Z 306.019,A -85,B 0,C 180,E1 -12973.899,E2 -12973.899} C_VEL
LIN {X 0,Y 361.967,Z 306.017,A -85,B 0,C 180,E1 -12977.938,E2 -12977.938} C_VEL
LIN {X 0,Y 361.86,Z 306.021,A -85,B 0,C 180,E1 -12981.655,E2 -12981.655} C_VEL
LIN {X 0,Y 361.882,Z 306.027,A -85,B 0,C 180,E1 -12985.293,E2 -12985.293} C_VEL
LIN {X 0,Y 361.854,Z 306.036,A -85,B 0,C 180,E1 -12989.074,E2 -12989.074} C_VEL
LIN {X 0,Y 361.848,Z 306.036,A -85,B 0,C 180,E1 -12992.945,E2 -12992.945} C_VEL
LIN {X 0,Y 361.867,Z 306.035,A -85,B 0,C 180,E1 -12995.637,E2 -12995.637} C_VEL
LIN {X 0,Y 361.9,Z 306.095,A -85,B 0,C 180,E1 -12999.389,E2 -12999.389} C_VEL
LIN {X 0,Y 364.193,Z 315.978,A -85,B 0,C 180,E1 -13003.261,E2 -13003.261} C_VEL
LIN {X 0,Y 366.517,Z 325.604,A -85,B 0,C 180,E1 -13006.774,E2 -13006.774} C_VEL
LIN {X 0,Y 369.068,Z 336.333,A -85,B 0,C 180,E1 -13010.423,E2 -13010.423} C_VEL
LIN {X 0,Y 370.714,Z 343.623,A -85,B 0,C 180,E1 -13012.772,E2 -13012.772} C_VEL
LIN {X 0,Y 369.492,Z 351.03,A -85,B 0,C 180,E1 -13014.874,E2 -13014.874} C_VEL
LIN {X 0,Y 366.95,Z 365.464,A -85,B 0,C 180,E1 -13018.861,E2 -13018.861} C_VEL
LIN {X 0,Y 365.391,Z 376.194,A -85,B 0,C 180,E1 -13021.79,E2 -13021.79} C_VEL
LIN {X 0,Y 369.65,Z 399.496,A -85,B 0,C 180,E1 -13022.711,E2 -13022.711} C_VEL
LIN {X 0,Y 371.738,Z 414.643,A -85,B 0,C 180,E1 -13023.476,E2 -13023.476} C_VEL
LIN {X 0,Y 372.692,Z 426.321,A -85,B 0,C 180,E1 -13024.172,E2 -13024.172} C_VEL
LIN {X 0,Y 372.802,Z 433.83,A -85,B 0,C 180,E1 -13024.663,E2 -13024.663} C_VEL
LIN {X 0,Y 371.361,Z 446.546,A -85,B 0,C 180,E1 -13025.545,E2 -13025.545} C_VEL
LIN {X 0,Y 369.481,Z 460.613,A -85,B 0,C 180,E1 -13026.753,E2 -13026.753} C_VEL
LIN {X 0,Y 367.667,Z 473.401,A -85,B 0,C 180,E1 -13028.115,E2 -13028.115} C_VEL
LIN {X 0,Y 366.189,Z 484.155,A -85,B 0,C 180,E1 -13029.497,E2 -13029.497} C_VEL
LIN {X 0,Y 364.668,Z 495.098,A -85,B 0,C 180,E1 -13031.167,E2 -13031.167} C_VEL
LIN {X 0,Y 363.176,Z 505.76,A -85,B 0,C 180,E1 -13033.126,E2 -13033.126} C_VEL
LIN {X 0,Y 362.137,Z 514.641,A -85,B 0,C 180,E1 -13035.1,E2 -13035.1} C_VEL
LIN {X 0,Y 361.326,Z 522.039,A -85,B 0,C 180,E1 -13037.075,E2 -13037.075} C_VEL
LIN {X 0,Y 360.872,Z 528.919,A -85,B 0,C 180,E1 -13039.338,E2 -13039.338} C_VEL
LIN {X 0,Y 360.651,Z 534.309,A -85,B 0,C 180,E1 -13041.596,E2 -13041.596} C_VEL
LIN {X 0,Y 360.757,Z 537.753,A -85,B 0,C 180,E1 -13043.485,E2 -13043.485} C_VEL
LIN {X 0,Y 360.699,Z 540.468,A -85,B 0,C 180,E1 -13045.53,E2 -13045.53} C_VEL
LIN {X 0,Y 360.852,Z 541.541,A -85,B 0,C 180,E1 -13046.651,E2 -13046.651} C_VEL
LIN {X 0,Y 360.894,Z 542.764,A -85,B 0,C 180,E1 -13048.884,E2 -13048.884} C_VEL
LIN {X 0,Y 360.894,Z 542.763,A -85,B 0,C 180,E1 -13051.116,E2 -13051.116} C_VEL
LIN {X 0,Y 360.874,Z 541.541,A -85,B 0,C 180,E1 -13053.35,E2 -13053.35} C_VEL
LIN {X 0,Y 360.782,Z 539.103,A -85,B 0,C 180,E1 -13055.59,E2 -13055.59} C_VEL
LIN {X 0,Y 360.696,Z 535.399,A -85,B 0,C 180,E1 -13057.839,E2 -13057.839} C_VEL
LIN {X 0,Y 360.798,Z 530.362,A -85,B 0,C 180,E1 -13060.097,E2 -13060.097} C_VEL
LIN {X 0,Y 361.205,Z 523.874,A -85,B 0,C 180,E1 -13062.359,E2 -13062.359} C_VEL
LIN {X 0,Y 362.005,Z 515.748,A -85,B 0,C 180,E1 -13064.619,E2 -13064.619} C_VEL
LIN {X 0,Y 362.955,Z 507.087,A -85,B 0,C 180,E1 -13066.596,E2 -13066.596} C_VEL
LIN {X 0,Y 364.247,Z 498.343,A -85,B 0,C 180,E1 -13068.273,E2 -13068.273} C_VEL
LIN {X 0,Y 365.68,Z 487.703,A -85,B 0,C 180,E1 -13069.992,E2 -13069.992} C_VEL
LIN {X 0,Y 367.419,Z 475.658,A -85,B 0,C 180,E1 -13071.606,E2 -13071.606} C_VEL
LIN {X 0,Y 369.128,Z 463.305,A -85,B 0,C 180,E1 -13072.974,E2 -13072.974} C_VEL
LIN {X 0,Y 370.924,Z 449.868,A -85,B 0,C 180,E1 -13074.188,E2 -13074.188} C_VEL
LIN {X 0,Y 372.544,Z 435.921,A -85,B 0,C 180,E1 -13075.197,E2 -13075.197} C_VEL
LIN {X 0,Y 372.885,Z 430.163,A -85,B 0,C 180,E1 -13075.56,E2 -13075.56} C_VEL
LIN {X 0,Y 372.74,Z 411.394,A -85,B 0,C 180,E1 -13076.999,E2 -13076.999} C_VEL
LIN {X 0,Y 371.607,Z 398.02,A -85,B 0,C 180,E1 -13077.982,E2 -13077.982} C_VEL
LIN {X 0,Y 369.167,Z 384.805,A -85,B 0,C 180,E1 -13078.985,E2 -13078.985} C_VEL
LIN {X 0,Y 366.715,Z 374.076,A -85,B 0,C 180,E1 -13079.851,E2 -13079.851} C_VEL
LIN {X 0,Y 369.316,Z 362.464,A -85,B 0,C 180,E1 -13083.495,E2 -13083.495} C_VEL
LIN {X 0,Y 372.6,Z 352.179,A -85,B 0,C 180,E1 -13087.128,E2 -13087.128} C_VEL
LIN {X 0,Y 372.806,Z 350.916,A -85,B 0,C 180,E1 -13087.649,E2 -13087.649} C_VEL
LIN {X 0,Y 371.858,Z 346.422,A -85,B 0,C 180,E1 -13089.986,E2 -13089.986} C_VEL
LIN {X 0,Y 370.827,Z 342.699,A -85,B 0,C 180,E1 -13092.342,E2 -13092.342} C_VEL
LIN {X 0,Y 369.702,Z 339.026,A -85,B 0,C 180,E1 -13095.302,E2 -13095.302} C_VEL
LIN {X 0,Y 368.773,Z 336.451,A -85,B 0,C 180,E1 -13098.162,E2 -13098.162} C_VEL
LIN {X 0,Y 367.905,Z 334.479,A -85,B 0,C 180,E1 -13101.556,E2 -13101.556} C_VEL
LIN {X 0,Y 367.399,Z 333.798,A -85,B 0,C 180,E1 -13103.63,E2 -13103.63} C_VEL
LIN {X 0,Y 366.658,Z 333.478,A -85,B 0,C 180,E1 -13106.23,E2 -13106.23} C_VEL
LIN {X 0,Y 365.829,Z 333.697,A -85,B 0,C 180,E1 -13109.827,E2 -13109.827} C_VEL
LIN {X 0,Y 365.138,Z 334.645,A -85,B 0,C 180,E1 -13113.724,E2 -13113.724} C_VEL
LIN {X 0,Y 364.965,Z 335.196,A -85,B 0,C 180,E1 -13115.239,E2 -13115.239} C_VEL
LIN {X 0,Y 366.343,Z 338.035,A -85,B 0,C 180,E1 -13115.678,E2 -13115.678} C_VEL
LIN {X 0,Y 370.345,Z 344.747,A -85,B 0,C 180,E1 -13116.844,E2 -13116.844} C_VEL
LIN {X 0,Y 374.497,Z 353.648,A -85,B 0,C 180,E1 -13118.22,E2 -13118.22} C_VEL
LIN {X 0,Y 377.136,Z 360.782,A -85,B 0,C 180,E1 -13119.264,E2 -13119.264} C_VEL
LIN {X 0,Y 375.494,Z 373.155,A -85,B 0,C 180,E1 -13120.454,E2 -13120.454} C_VEL
LIN {X 0,Y 373.382,Z 385.618,A -85,B 0,C 180,E1 -13121.906,E2 -13121.906} C_VEL
LIN {X 0,Y 371.741,Z 394.958,A -85,B 0,C 180,E1 -13123.243,E2 -13123.243} C_VEL
LIN {X 0,Y 369.985,Z 404.264,A -85,B 0,C 180,E1 -13124.86,E2 -13124.86} C_VEL
LIN {X 0,Y 368.088,Z 413.181,A -85,B 0,C 180,E1 -13126.755,E2 -13126.755} C_VEL
LIN {X 0,Y 366.75,Z 419.31,A -85,B 0,C 180,E1 -13128.392,E2 -13128.392} C_VEL
LIN {X 0,Y 365.593,Z 424.268,A -85,B 0,C 180,E1 -13130.037,E2 -13130.037} C_VEL
LIN {X 0,Y 364.628,Z 428.196,A -85,B 0,C 180,E1 -13131.688,E2 -13131.688} C_VEL
LIN {X 0,Y 363.733,Z 431.146,A -85,B 0,C 180,E1 -13133.343,E2 -13133.343} C_VEL
LIN {X 0,Y 363.398,Z 432.569,A -85,B 0,C 180,E1 -13134.451,E2 -13134.451} C_VEL
LIN {X 0,Y 363.143,Z 433.583,A -85,B 0,C 180,E1 -13135.56,E2 -13135.56} C_VEL
LIN {X 0,Y 362.508,Z 434.471,A -85,B 0,C 180,E1 -13137.778,E2 -13137.778} C_VEL
LIN {X 0,Y 362.345,Z 434.33,A -85,B 0,C 180,E1 -13138.889,E2 -13138.889} C_VEL
LIN {X 0,Y 362.091,Z 433.821,A -85,B 0,C 180,E1 -13140,E2 -13140} C_VEL
LIN {X 0,Y 362.054,Z 432.858,A -85,B 0,C 180,E1 -13141.112,E2 -13141.112} C_VEL
LIN {X 0,Y 361.932,Z 431.51,A -85,B 0,C 180,E1 -13142.226,E2 -13142.226} C_VEL
LIN {X 0,Y 361.898,Z 428.716,A -85,B 0,C 180,E1 -13143.897,E2 -13143.897} C_VEL
LIN {X 0,Y 362.201,Z 424.922,A -85,B 0,C 180,E1 -13145.568,E2 -13145.568} C_VEL
LIN {X 0,Y 362.561,Z 419.794,A -85,B 0,C 180,E1 -13147.324,E2 -13147.324} C_VEL
LIN {X 0,Y 363.005,Z 413.265,A -85,B 0,C 180,E1 -13149.106,E2 -13149.106} C_VEL
LIN {X 0,Y 363.568,Z 405.327,A -85,B 0,C 180,E1 -13150.864,E2 -13150.864} C_VEL
LIN {X 0,Y 364.171,Z 396.057,A -85,B 0,C 180,E1 -13152.539,E2 -13152.539} C_VEL
LIN {X 0,Y 365.104,Z 384.702,A -85,B 0,C 180,E1 -13154.207,E2 -13154.207} C_VEL
LIN {X 0,Y 365.97,Z 373.046,A -85,B 0,C 180,E1 -13155.596,E2 -13155.596} C_VEL
LIN {X 0,Y 366.787,Z 360.161,A -85,B 0,C 180,E1 -13156.847,E2 -13156.847} C_VEL
LIN {X 0,Y 367.667,Z 346.554,A -85,B 0,C 180,E1 -13157.881,E2 -13157.881} C_VEL
LIN {X 0,Y 367.517,Z 343.396,A -85,B 0,C 180,E1 -13158.105,E2 -13158.105} C_VEL
LIN {X 0,Y 363.819,Z 328.665,A -85,B 0,C 180,E1 -13159.096,E2 -13159.096} C_VEL
LIN {X 0,Y 361.28,Z 318.653,A -85,B 0,C 180,E1 -13159.635,E2 -13159.635} C_VEL
LIN {X 0,Y 361.265,Z 315.113,A -85,B 0,C 180,E1 -13162.897,E2 -13162.897} C_VEL
LIN {X 0,Y 361.314,Z 311.218,A -85,B 0,C 180,E1 -13166.576,E2 -13166.576} C_VEL
LIN {X 0,Y 361.332,Z 307.32,A -85,B 0,C 180,E1 -13170.378,E2 -13170.378} C_VEL
LIN {X 0,Y 361.353,Z 306.101,A -85,B 0,C 180,E1 -13171.677,E2 -13171.677} C_VEL
LIN {X 0,Y 361.728,Z 306.053,A -85,B 0,C 180,E1 -13175.311,E2 -13175.311} C_VEL
LIN {X 0,Y 361.864,Z 306.035,A -85,B 0,C 180,E1 -13178.425,E2 -13178.425} C_VEL
LIN {X 0,Y 361.829,Z 306.034,A -85,B 0,C 180,E1 -13181.331,E2 -13181.331} C_VEL
LIN {X 0,Y 361.865,Z 306.119,A -85,B 0,C 180,E1 -13184.861,E2 -13184.861} C_VEL
LIN {X 0,Y 362.399,Z 309.421,A -85,B 0,C 180,E1 -13187.471,E2 -13187.471} C_VEL
LIN {X 0,Y 362.585,Z 312.964,A -85,B 0,C 180,E1 -13190.235,E2 -13190.235} C_VEL
LIN {X 0,Y 362.548,Z 316.676,A -85,B 0,C 180,E1 -13193.063,E2 -13193.063} C_VEL
LIN {X 0,Y 362.458,Z 321.321,A -85,B 0,C 180,E1 -13196.487,E2 -13196.487} C_VEL
LIN {X 0,Y 362.45,Z 325.938,A -85,B 0,C 180,E1 -13199.725,E2 -13199.725} C_VEL
LIN {X 0,Y 362.491,Z 328.896,A -85,B 0,C 180,E1 -13201.539,E2 -13201.539} C_VEL
LIN {X 0,Y 368.991,Z 344.68,A -85,B 0,C 180,E1 -13202.546,E2 -13202.546} C_VEL
LIN {X 0,Y 374.074,Z 359.151,A -85,B 0,C 180,E1 -13203.604,E2 -13203.604} C_VEL
LIN {X 0,Y 375.768,Z 365.042,A -85,B 0,C 180,E1 -13204.066,E2 -13204.066} C_VEL
LIN {X 0,Y 375.866,Z 368.222,A -85,B 0,C 180,E1 -13204.265,E2 -13204.265} C_VEL
LIN {X 0,Y 374.824,Z 380.908,A -85,B 0,C 180,E1 -13205.077,E2 -13205.077} C_VEL
LIN {X 0,Y 373.445,Z 394.18,A -85,B 0,C 180,E1 -13206.133,E2 -13206.133} C_VEL
LIN {X 0,Y 371.649,Z 407.951,A -85,B 0,C 180,E1 -13207.484,E2 -13207.484} C_VEL
LIN {X 0,Y 369.959,Z 420.346,A -85,B 0,C 180,E1 -13208.988,E2 -13208.988} C_VEL
LIN {X 0,Y 368.425,Z 430.721,A -85,B 0,C 180,E1 -13210.499,E2 -13210.499} C_VEL
LIN {X 0,Y 366.849,Z 440.319,A -85,B 0,C 180,E1 -13212.15,E2 -13212.15} C_VEL
LIN {X 0,Y 365.405,Z 448.74,A -85,B 0,C 180,E1 -13213.863,E2 -13213.863} C_VEL
LIN {X 0,Y 364.07,Z 457.476,A -85,B 0,C 180,E1 -13216.036,E2 -13216.036} C_VEL
LIN {X 0,Y 362.888,Z 464.719,A -85,B 0,C 180,E1 -13218.267,E2 -13218.267} C_VEL
LIN {X 0,Y 362.072,Z 470.449,A -85,B 0,C 180,E1 -13220.503,E2 -13220.503} C_VEL
LIN {X 0,Y 361.556,Z 474.341,A -85,B 0,C 180,E1 -13222.459,E2 -13222.459} C_VEL
LIN {X 0,Y 361.145,Z 477.276,A -85,B 0,C 180,E1 -13224.416,E2 -13224.416} C_VEL
LIN {X 0,Y 361.045,Z 479.532,A -85,B 0,C 180,E1 -13226.652,E2 -13226.652} C_VEL
LIN {X 0,Y 360.826,Z 480.693,A -85,B 0,C 180,E1 -13228.884,E2 -13228.884} C_VEL
LIN {X 0,Y 360.826,Z 480.706,A -85,B 0,C 180,E1 -13231.116,E2 -13231.116} C_VEL
LIN {X 0,Y 361.021,Z 479.599,A -85,B 0,C 180,E1 -13233.348,E2 -13233.348} C_VEL
LIN {X 0,Y 361.144,Z 477.397,A -85,B 0,C 180,E1 -13235.584,E2 -13235.584} C_VEL
LIN {X 0,Y 361.617,Z 474.015,A -85,B 0,C 180,E1 -13237.819,E2 -13237.819} C_VEL
LIN {X 0,Y 362.222,Z 469.382,A -85,B 0,C 180,E1 -13240.056,E2 -13240.056} C_VEL
LIN {X 0,Y 363.147,Z 463.353,A -85,B 0,C 180,E1 -13242.291,E2 -13242.291} C_VEL
LIN {X 0,Y 364.374,Z 455.758,A -85,B 0,C 180,E1 -13244.521,E2 -13244.521} C_VEL
LIN {X 0,Y 365.588,Z 447.789,A -85,B 0,C 180,E1 -13246.443,E2 -13246.443} C_VEL
LIN {X 0,Y 367.244,Z 437.86,A -85,B 0,C 180,E1 -13248.407,E2 -13248.407} C_VEL
LIN {X 0,Y 368.873,Z 427.839,A -85,B 0,C 180,E1 -13250.056,E2 -13250.056} C_VEL
LIN {X 0,Y 370.479,Z 416.391,A -85,B 0,C 180,E1 -13251.638,E2 -13251.638} C_VEL
LIN {X 0,Y 372.28,Z 403.781,A -85,B 0,C 180,E1 -13253.062,E2 -13253.062} C_VEL
LIN {X 0,Y 373.894,Z 390.613,A -85,B 0,C 180,E1 -13254.279,E2 -13254.279} C_VEL
LIN {X 0,Y 375.313,Z 375.971,A -85,B 0,C 180,E1 -13255.363,E2 -13255.363} C_VEL
LIN {X 0,Y 376.012,Z 367.02,A -85,B 0,C 180,E1 -13255.9,E2 -13255.9} C_VEL
LIN {X 0,Y 375.61,Z 364.445,A -85,B 0,C 180,E1 -13256.087,E2 -13256.087} C_VEL
LIN {X 0,Y 371.402,Z 351.22,A -85,B 0,C 180,E1 -13257.098,E2 -13257.098} C_VEL
LIN {X 0,Y 369.74,Z 348.102,A -85,B 0,C 180,E1 -13257.373,E2 -13257.373} C_VEL
LIN {X 0,Y 365.422,Z 344.16,A -85,B 0,C 180,E1 -13257.89,E2 -13257.89} C_VEL
LIN {X 0,Y 360.892,Z 340.291,A -85,B 0,C 180,E1 -13258.411,E2 -13258.411} C_VEL
LIN {X 0,Y 358.861,Z 337.255,A -85,B 0,C 180,E1 -13258.679,E2 -13258.679} C_VEL
LIN {X 0,Y 355.554,Z 329.3,A -85,B 0,C 180,E1 -13259.193,E2 -13259.193} C_VEL
LIN {X 0,Y 355.474,Z 324.747,A -85,B 0,C 180,E1 -13262.263,E2 -13262.263} C_VEL
LIN {X 0,Y 355.551,Z 319.8,A -85,B 0,C 180,E1 -13265.862,E2 -13265.862} C_VEL
LIN {X 0,Y 355.627,Z 314.874,A -85,B 0,C 180,E1 -13269.58,E2 -13269.58} C_VEL
LIN {X 0,Y 355.497,Z 311.536,A -85,B 0,C 180,E1 -13272.234,E2 -13272.234} C_VEL
LIN {X 0,Y 355.106,Z 308.576,A -85,B 0,C 180,E1 -13274.562,E2 -13274.562} C_VEL
LIN {X 0,Y 354.791,Z 306.921,A -85,B 0,C 180,E1 -13275.948,E2 -13275.948} C_VEL
LIN {X 0,Y 354.787,Z 306.915,A -85,B 0,C 180,E1 -13279.179,E2 -13279.179} C_VEL
LIN {X 0,Y 354.806,Z 306.915,A -85,B 0,C 180,E1 -13282.403,E2 -13282.403} C_VEL
LIN {X 0,Y 354.812,Z 306.916,A -85,B 0,C 180,E1 -13284.941,E2 -13284.941} C_VEL
LIN {X 0,Y 354.793,Z 306.918,A -85,B 0,C 180,E1 -13288.405,E2 -13288.405} C_VEL
LIN {X 0,Y 354.796,Z 306.915,A -85,B 0,C 180,E1 -13291.614,E2 -13291.614} C_VEL
LIN {X 0,Y 354.834,Z 306.912,A -85,B 0,C 180,E1 -13295.657,E2 -13295.657} C_VEL
LIN {X 0,Y 354.827,Z 306.902,A -85,B 0,C 180,E1 -13299.113,E2 -13299.113} C_VEL
LIN {X 0,Y 354.88,Z 306.89,A -85,B 0,C 180,E1 -13302.719,E2 -13302.719} C_VEL
LIN {X 0,Y 354.952,Z 306.896,A -85,B 0,C 180,E1 -13306.255,E2 -13306.255} C_VEL
LIN {X 0,Y 354.956,Z 306.888,A -85,B 0,C 180,E1 -13309.735,E2 -13309.735} C_VEL
LIN {X 0,Y 355.089,Z 306.864,A -85,B 0,C 180,E1 -13313.18,E2 -13313.18} C_VEL
LIN {X 0,Y 355.243,Z 306.857,A -85,B 0,C 180,E1 -13317.732,E2 -13317.732} C_VEL
LIN {X 0,Y 355.375,Z 306.824,A -85,B 0,C 180,E1 -13320,E2 -13320} C_VEL
LIN {X 0,Y 355.233,Z 306.862,A -85,B 0,C 180,E1 -13322.268,E2 -13322.268} C_VEL
LIN {X 0,Y 355.105,Z 306.869,A -85,B 0,C 180,E1 -13326.82,E2 -13326.82} C_VEL
LIN {X 0,Y 354.956,Z 306.879,A -85,B 0,C 180,E1 -13330.265,E2 -13330.265} C_VEL
LIN {X 0,Y 354.943,Z 306.897,A -85,B 0,C 180,E1 -13334.019,E2 -13334.019} C_VEL
LIN {X 0,Y 354.922,Z 306.896,A -85,B 0,C 180,E1 -13338.108,E2 -13338.108} C_VEL
LIN {X 0,Y 354.814,Z 306.899,A -85,B 0,C 180,E1 -13342.107,E2 -13342.107} C_VEL
LIN {X 0,Y 354.848,Z 306.909,A -85,B 0,C 180,E1 -13344.577,E2 -13344.577} C_VEL
LIN {X 0,Y 354.8,Z 306.914,A -85,B 0,C 180,E1 -13348.385,E2 -13348.385} C_VEL
LIN {X 0,Y 354.786,Z 306.916,A -85,B 0,C 180,E1 -13352.333,E2 -13352.333} C_VEL
LIN {X 0,Y 354.821,Z 306.912,A -85,B 0,C 180,E1 -13355.699,E2 -13355.699} C_VEL
LIN {X 0,Y 354.824,Z 307.007,A -85,B 0,C 180,E1 -13358.785,E2 -13358.785} C_VEL
LIN {X 0,Y 357.119,Z 316.666,A -85,B 0,C 180,E1 -13362.687,E2 -13362.687} C_VEL
LIN {X 0,Y 359.414,Z 326.445,A -85,B 0,C 180,E1 -13366.344,E2 -13366.344} C_VEL
LIN {X 0,Y 361.762,Z 336.083,A -85,B 0,C 180,E1 -13369.733,E2 -13369.733} C_VEL
LIN {X 0,Y 363.657,Z 344.148,A -85,B 0,C 180,E1 -13372.407,E2 -13372.407} C_VEL
LIN {X 0,Y 363.565,Z 346.71,A -85,B 0,C 180,E1 -13373.184,E2 -13373.184} C_VEL
LIN {X 0,Y 361.11,Z 359.365,A -85,B 0,C 180,E1 -13376.811,E2 -13376.811} C_VEL
LIN {X 0,Y 358.864,Z 373.157,A -85,B 0,C 180,E1 -13380.686,E2 -13380.686} C_VEL
LIN {X 0,Y 358.611,Z 374.928,A -85,B 0,C 180,E1 -13381.185,E2 -13381.185} C_VEL
LIN {X 0,Y 363.052,Z 399.248,A -85,B 0,C 180,E1 -13382.183,E2 -13382.183} C_VEL
LIN {X 0,Y 365.16,Z 414.948,A -85,B 0,C 180,E1 -13383.004,E2 -13383.004} C_VEL
LIN {X 0,Y 366.171,Z 427.785,A -85,B 0,C 180,E1 -13383.804,E2 -13383.804} C_VEL
LIN {X 0,Y 366.3,Z 433.784,A -85,B 0,C 180,E1 -13384.217,E2 -13384.217} C_VEL
LIN {X 0,Y 364.648,Z 447.727,A -85,B 0,C 180,E1 -13385.216,E2 -13385.216} C_VEL
LIN {X 0,Y 362.705,Z 461.45,A -85,B 0,C 180,E1 -13386.444,E2 -13386.444} C_VEL
LIN {X 0,Y 360.835,Z 473.981,A -85,B 0,C 180,E1 -13387.83,E2 -13387.83} C_VEL
LIN {X 0,Y 359.164,Z 485.52,A -85,B 0,C 180,E1 -13389.377,E2 -13389.377} C_VEL
LIN {X 0,Y 357.599,Z 496.137,A -85,B 0,C 180,E1 -13391.078,E2 -13391.078} C_VEL
LIN {X 0,Y 356.087,Z 506.524,A -85,B 0,C 180,E1 -13393.075,E2 -13393.075} C_VEL
LIN {X 0,Y 355.025,Z 515.165,A -85,B 0,C 180,E1 -13395.088,E2 -13395.088} C_VEL
LIN {X 0,Y 354.152,Z 523.283,A -85,B 0,C 180,E1 -13397.392,E2 -13397.392} C_VEL
LIN {X 0,Y 353.698,Z 529.771,A -85,B 0,C 180,E1 -13399.699,E2 -13399.699} C_VEL
LIN {X 0,Y 353.579,Z 534.801,A -85,B 0,C 180,E1 -13402.002,E2 -13402.002} C_VEL
LIN {X 0,Y 353.682,Z 537.354,A -85,B 0,C 180,E1 -13403.486,E2 -13403.486} C_VEL
LIN {X 0,Y 353.622,Z 539.858,A -85,B 0,C 180,E1 -13405.441,E2 -13405.441} C_VEL
LIN {X 0,Y 353.806,Z 541.693,A -85,B 0,C 180,E1 -13407.723,E2 -13407.723} C_VEL
LIN {X 0,Y 353.811,Z 542.313,A -85,B 0,C 180,E1 -13410,E2 -13410} C_VEL
LIN {X 0,Y 353.831,Z 541.694,A -85,B 0,C 180,E1 -13412.277,E2 -13412.277} C_VEL
LIN {X 0,Y 353.666,Z 539.858,A -85,B 0,C 180,E1 -13414.559,E2 -13414.559} C_VEL
LIN {X 0,Y 353.677,Z 536.802,A -85,B 0,C 180,E1 -13416.848,E2 -13416.848} C_VEL
LIN {X 0,Y 353.656,Z 532.439,A -85,B 0,C 180,E1 -13419.148,E2 -13419.148} C_VEL
LIN {X 0,Y 353.953,Z 526.695,A -85,B 0,C 180,E1 -13421.453,E2 -13421.453} C_VEL
LIN {X 0,Y 354.548,Z 519.412,A -85,B 0,C 180,E1 -13423.761,E2 -13423.761} C_VEL
LIN {X 0,Y 355.432,Z 511.626,A -85,B 0,C 180,E1 -13425.776,E2 -13425.776} C_VEL
LIN {X 0,Y 356.745,Z 502.275,A -85,B 0,C 180,E1 -13427.78,E2 -13427.78} C_VEL
LIN {X 0,Y 358.319,Z 491.438,A -85,B 0,C 180,E1 -13429.701,E2 -13429.701} C_VEL
LIN {X 0,Y 359.975,Z 480.457,A -85,B 0,C 180,E1 -13431.323,E2 -13431.323} C_VEL
LIN {X 0,Y 361.749,Z 467.894,A -85,B 0,C 180,E1 -13432.865,E2 -13432.865} C_VEL
LIN {X 0,Y 363.822,Z 454.033,A -85,B 0,C 180,E1 -13434.236,E2 -13434.236} C_VEL
LIN {X 0,Y 365.568,Z 439.8,A -85,B 0,C 180,E1 -13435.369,E2 -13435.369} C_VEL
LIN {X 0,Y 366.374,Z 432.374,A -85,B 0,C 180,E1 -13435.889,E2 -13435.889} C_VEL
LIN {X 0,Y 366.753,Z 416.952,A -85,B 0,C 180,E1 -13437.204,E2 -13437.204} C_VEL
LIN {X 0,Y 366.1,Z 402.689,A -85,B 0,C 180,E1 -13438.324,E2 -13438.324} C_VEL
LIN {X 0,Y 364.161,Z 389.577,A -85,B 0,C 180,E1 -13439.377,E2 -13439.377} C_VEL
LIN {X 0,Y 361.206,Z 376.769,A -85,B 0,C 180,E1 -13440.481,E2 -13440.481} C_VEL
LIN {X 0,Y 360.37,Z 372.841,A -85,B 0,C 180,E1 -13440.83,E2 -13440.83} C_VEL
LIN {X 0,Y 362.909,Z 362.677,A -85,B 0,C 180,E1 -13444.167,E2 -13444.167} C_VEL
LIN {X 0,Y 365.78,Z 354.228,A -85,B 0,C 180,E1 -13447.246,E2 -13447.246} C_VEL
LIN {X 0,Y 365.956,Z 352.393,A -85,B 0,C 180,E1 -13448.058,E2 -13448.058} C_VEL
LIN {X 0,Y 365.063,Z 348.426,A -85,B 0,C 180,E1 -13450.201,E2 -13450.201} C_VEL
LIN {X 0,Y 363.95,Z 344.478,A -85,B 0,C 180,E1 -13452.795,E2 -13452.795} C_VEL
LIN {X 0,Y 362.875,Z 340.922,A -85,B 0,C 180,E1 -13455.795,E2 -13455.795} C_VEL
LIN {X 0,Y 361.766,Z 338.07,A -85,B 0,C 180,E1 -13459.258,E2 -13459.258} C_VEL
LIN {X 0,Y 361.215,Z 336.841,A -85,B 0,C 180,E1 -13461.493,E2 -13461.493} C_VEL
LIN {X 0,Y 360.481,Z 335.957,A -85,B 0,C 180,E1 -13464.205,E2 -13464.205} C_VEL
LIN {X 0,Y 359.656,Z 335.649,A -85,B 0,C 180,E1 -13467.168,E2 -13467.168} C_VEL
LIN {X 0,Y 358.837,Z 335.954,A -85,B 0,C 180,E1 -13470.683,E2 -13470.683} C_VEL
LIN {X 0,Y 358.316,Z 336.952,A -85,B 0,C 180,E1 -13474.157,E2 -13474.157} C_VEL
LIN {X 0,Y 359.275,Z 339.084,A -85,B 0,C 180,E1 -13474.51,E2 -13474.51} C_VEL
LIN {X 0,Y 360.713,Z 340.707,A -85,B 0,C 180,E1 -13474.908,E2 -13474.908} C_VEL
LIN {X 0,Y 366.1,Z 350.646,A -85,B 0,C 180,E1 -13476.698,E2 -13476.698} C_VEL
LIN {X 0,Y 369.398,Z 358.293,A -85,B 0,C 180,E1 -13477.949,E2 -13477.949} C_VEL
LIN {X 0,Y 371.27,Z 363.653,A -85,B 0,C 180,E1 -13478.793,E2 -13478.793} C_VEL
LIN {X 0,Y 369.293,Z 376.741,A -85,B 0,C 180,E1 -13480.112,E2 -13480.112} C_VEL
LIN {X 0,Y 367.426,Z 386.663,A -85,B 0,C 180,E1 -13481.314,E2 -13481.314} C_VEL
LIN {X 0,Y 365.329,Z 397.634,A -85,B 0,C 180,E1 -13482.94,E2 -13482.94} C_VEL
LIN {X 0,Y 363.481,Z 406.645,A -85,B 0,C 180,E1 -13484.582,E2 -13484.582} C_VEL
LIN {X 0,Y 361.58,Z 414.703,A -85,B 0,C 180,E1 -13486.373,E2 -13486.373} C_VEL
LIN {X 0,Y 360.044,Z 421.224,A -85,B 0,C 180,E1 -13488.173,E2 -13488.173} C_VEL
LIN {X 0,Y 358.821,Z 426.035,A -85,B 0,C 180,E1 -13489.847,E2 -13489.847} C_VEL
LIN {X 0,Y 357.792,Z 429.791,A -85,B 0,C 180,E1 -13491.528,E2 -13491.528} C_VEL
LIN {X 0,Y 356.85,Z 432.616,A -85,B 0,C 180,E1 -13493.214,E2 -13493.214} C_VEL
LIN {X 0,Y 356.487,Z 433.973,A -85,B 0,C 180,E1 -13494.343,E2 -13494.343} C_VEL
LIN {X 0,Y 356.188,Z 434.901,A -85,B 0,C 180,E1 -13495.473,E2 -13495.473} C_VEL
LIN {X 0,Y 355.529,Z 435.656,A -85,B 0,C 180,E1 -13497.734,E2 -13497.734} C_VEL
LIN {X 0,Y 355.354,Z 435.449,A -85,B 0,C 180,E1 -13498.867,E2 -13498.867} C_VEL
LIN {X 0,Y 355.068,Z 434.863,A -85,B 0,C 180,E1 -13500,E2 -13500} C_VEL
LIN {X 0,Y 355.029,Z 433.829,A -85,B 0,C 180,E1 -13501.134,E2 -13501.134} C_VEL
LIN {X 0,Y 354.905,Z 432.418,A -85,B 0,C 180,E1 -13502.27,E2 -13502.27} C_VEL
LIN {X 0,Y 354.868,Z 429.522,A -85,B 0,C 180,E1 -13503.975,E2 -13503.975} C_VEL
LIN {X 0,Y 355.194,Z 425.607,A -85,B 0,C 180,E1 -13505.678,E2 -13505.678} C_VEL
LIN {X 0,Y 355.539,Z 420.648,A -85,B 0,C 180,E1 -13507.382,E2 -13507.382} C_VEL
LIN {X 0,Y 355.985,Z 414.06,A -85,B 0,C 180,E1 -13509.203,E2 -13509.203} C_VEL
LIN {X 0,Y 356.603,Z 405.674,A -85,B 0,C 180,E1 -13511.079,E2 -13511.079} C_VEL
LIN {X 0,Y 357.237,Z 396.239,A -85,B 0,C 180,E1 -13512.787,E2 -13512.787} C_VEL
LIN {X 0,Y 358.116,Z 385.758,A -85,B 0,C 180,E1 -13514.345,E2 -13514.345} C_VEL
LIN {X 0,Y 359.013,Z 374.144,A -85,B 0,C 180,E1 -13515.761,E2 -13515.761} C_VEL
LIN {X 0,Y 359.86,Z 361.309,A -85,B 0,C 180,E1 -13517.035,E2 -13517.035} C_VEL
LIN {X 0,Y 360.756,Z 347.847,A -85,B 0,C 180,E1 -13518.088,E2 -13518.088} C_VEL
LIN {X 0,Y 360.589,Z 344.505,A -85,B 0,C 180,E1 -13518.332,E2 -13518.332} C_VEL
LIN {X 0,Y 357.037,Z 330.282,A -85,B 0,C 180,E1 -13519.325,E2 -13519.325} C_VEL
LIN {X 0,Y 354.252,Z 319.205,A -85,B 0,C 180,E1 -13519.956,E2 -13519.956} C_VEL
LIN {X 0,Y 354.252,Z 314.695,A -85,B 0,C 180,E1 -13524.133,E2 -13524.133} C_VEL
LIN {X 0,Y 354.264,Z 311.571,A -85,B 0,C 180,E1 -13527.148,E2 -13527.148} C_VEL
LIN {X 0,Y 354.313,Z 307.57,A -85,B 0,C 180,E1 -13531.046,E2 -13531.046} C_VEL
LIN {X 0,Y 354.319,Z 307.147,A -85,B 0,C 180,E1 -13531.469,E2 -13531.469} C_VEL
LIN {X 0,Y 354.648,Z 306.933,A -85,B 0,C 180,E1 -13535.078,E2 -13535.078} C_VEL
LIN {X 0,Y 354.796,Z 306.915,A -85,B 0,C 180,E1 -13537.884,E2 -13537.884} C_VEL
LIN {X 0,Y 354.79,Z 306.911,A -85,B 0,C 180,E1 -13541.171,E2 -13541.171} C_VEL
LIN {X 0,Y 354.786,Z 307.004,A -85,B 0,C 180,E1 -13544.314,E2 -13544.314} C_VEL
LIN {X 0,Y 355.401,Z 310.402,A -85,B 0,C 180,E1 -13547.027,E2 -13547.027} C_VEL
LIN {X 0,Y 355.65,Z 313.247,A -85,B 0,C 180,E1 -13549.298,E2 -13549.298} C_VEL
LIN {X 0,Y 355.572,Z 317.086,A -85,B 0,C 180,E1 -13552.243,E2 -13552.243} C_VEL
LIN {X 0,Y 355.531,Z 320.792,A -85,B 0,C 180,E1 -13555.022,E2 -13555.022} C_VEL
LIN {X 0,Y 355.477,Z 325.277,A -85,B 0,C 180,E1 -13558.227,E2 -13558.227} C_VEL
LIN {X 0,Y 355.527,Z 329.327,A -85,B 0,C 180,E1 -13560.925,E2 -13560.925} C_VEL
LIN {X 0,Y 357.968,Z 335.171,A -85,B 0,C 180,E1 -13561.287,E2 -13561.287} C_VEL
LIN {X 0,Y 363.823,Z 349.602,A -85,B 0,C 180,E1 -13562.293,E2 -13562.293} C_VEL
LIN {X 0,Y 368.423,Z 363.605,A -85,B 0,C 180,E1 -13563.379,E2 -13563.379} C_VEL
LIN {X 0,Y 369.523,Z 367.585,A -85,B 0,C 180,E1 -13563.715,E2 -13563.715} C_VEL
LIN {X 0,Y 368.398,Z 381.854,A -85,B 0,C 180,E1 -13564.64,E2 -13564.64} C_VEL
LIN {X 0,Y 366.993,Z 394.776,A -85,B 0,C 180,E1 -13565.686,E2 -13565.686} C_VEL
LIN {X 0,Y 365.139,Z 408.55,A -85,B 0,C 180,E1 -13567.06,E2 -13567.06} C_VEL
LIN {X 0,Y 363.356,Z 420.95,A -85,B 0,C 180,E1 -13568.587,E2 -13568.587} C_VEL
LIN {X 0,Y 361.768,Z 431.326,A -85,B 0,C 180,E1 -13570.125,E2 -13570.125} C_VEL
LIN {X 0,Y 360.114,Z 440.925,A -85,B 0,C 180,E1 -13571.804,E2 -13571.804} C_VEL
LIN {X 0,Y 358.606,Z 449.348,A -85,B 0,C 180,E1 -13573.549,E2 -13573.549} C_VEL
LIN {X 0,Y 357.195,Z 458.085,A -85,B 0,C 180,E1 -13575.762,E2 -13575.762} C_VEL
LIN {X 0,Y 355.966,Z 465.327,A -85,B 0,C 180,E1 -13578.035,E2 -13578.035} C_VEL
LIN {X 0,Y 355.086,Z 471.059,A -85,B 0,C 180,E1 -13580.314,E2 -13580.314} C_VEL
LIN {X 0,Y 354.514,Z 475.118,A -85,B 0,C 180,E1 -13582.402,E2 -13582.402} C_VEL
LIN {X 0,Y 354.093,Z 477.886,A -85,B 0,C 180,E1 -13584.304,E2 -13584.304} C_VEL
LIN {X 0,Y 353.986,Z 480.14,A -85,B 0,C 180,E1 -13586.585,E2 -13586.585} C_VEL
LIN {X 0,Y 353.782,Z 481.299,A -85,B 0,C 180,E1 -13588.861,E2 -13588.861} C_VEL
LIN {X 0,Y 353.782,Z 481.312,A -85,B 0,C 180,E1 -13591.138,E2 -13591.138} C_VEL
LIN {X 0,Y 353.965,Z 480.206,A -85,B 0,C 180,E1 -13593.415,E2 -13593.415} C_VEL
LIN {X 0,Y 354.091,Z 478.006,A -85,B 0,C 180,E1 -13595.695,E2 -13595.695} C_VEL
LIN {X 0,Y 354.603,Z 474.622,A -85,B 0,C 180,E1 -13597.974,E2 -13597.974} C_VEL
LIN {X 0,Y 355.247,Z 469.989,A -85,B 0,C 180,E1 -13600.256,E2 -13600.256} C_VEL
LIN {X 0,Y 356.232,Z 463.959,A -85,B 0,C 180,E1 -13602.534,E2 -13602.534} C_VEL
LIN {X 0,Y 357.513,Z 456.364,A -85,B 0,C 180,E1 -13604.806,E2 -13604.806} C_VEL
LIN {X 0,Y 358.817,Z 448.261,A -85,B 0,C 180,E1 -13606.792,E2 -13606.792} C_VEL
LIN {X 0,Y 360.533,Z 438.46,A -85,B 0,C 180,E1 -13608.762,E2 -13608.762} C_VEL
LIN {X 0,Y 362.214,Z 428.438,A -85,B 0,C 180,E1 -13610.441,E2 -13610.441} C_VEL
LIN {X 0,Y 363.869,Z 417.276,A -85,B 0,C 180,E1 -13612.012,E2 -13612.012} C_VEL
LIN {X 0,Y 365.795,Z 404.369,A -85,B 0,C 180,E1 -13613.495,E2 -13613.495} C_VEL
LIN {X 0,Y 367.477,Z 391.194,A -85,B 0,C 180,E1 -13614.731,E2 -13614.731} C_VEL
LIN {X 0,Y 368.858,Z 377.537,A -85,B 0,C 180,E1 -13615.769,E2 -13615.769} C_VEL
LIN {X 0,Y 369.553,Z 367.544,A -85,B 0,C 180,E1 -13616.39,E2 -13616.39} C_VEL
LIN {X 0,Y 365.215,Z 353.51,A -85,B 0,C 180,E1 -13617.517,E2 -13617.517} C_VEL
LIN {X 0,Y 359.756,Z 339.3,A -85,B 0,C 180,E1 -13618.54,E2 -13618.54} C_VEL
LIN {X 0,Y 358.861,Z 337.255,A -85,B 0,C 180,E1 -13618.679,E2 -13618.679} C_VEL
LIN {X 0,Y 356.86,Z 334.225,A -85,B 0,C 180,E1 -13618.981,E2 -13618.981} C_VEL
LIN {X 0,Y 354.372,Z 332.014,A -85,B 0,C 180,E1 -13619.38,E2 -13619.38} C_VEL
LIN {X 0,Y 351.137,Z 329.948,A -85,B 0,C 180,E1 -13620.034,E2 -13620.034} C_VEL
LIN {X 0,Y 349.085,Z 328.607,A -85,B 0,C 180,E1 -13620.716,E2 -13620.716} C_VEL
LIN {X 0,Y 348.553,Z 327.767,A -85,B 0,C 180,E1 -13621.253,E2 -13621.253} C_VEL
LIN {X 0,Y 348.573,Z 323.318,A -85,B 0,C 180,E1 -13624.37,E2 -13624.37} C_VEL
LIN {X 0,Y 348.649,Z 318.262,A -85,B 0,C 180,E1 -13628.172,E2 -13628.172} C_VEL
LIN {X 0,Y 348.688,Z 315.673,A -85,B 0,C 180,E1 -13630.164,E2 -13630.164} C_VEL
LIN {X 0,Y 348.606,Z 313.641,A -85,B 0,C 180,E1 -13631.761,E2 -13631.761} C_VEL
LIN {X 0,Y 348.406,Z 311.61,A -85,B 0,C 180,E1 -13633.432,E2 -13633.432} C_VEL
LIN {X 0,Y 347.723,Z 307.8,A -85,B 0,C 180,E1 -13636.592,E2 -13636.592} C_VEL
LIN {X 0,Y 347.747,Z 307.792,A -85,B 0,C 180,E1 -13640.173,E2 -13640.173} C_VEL
LIN {X 0,Y 347.761,Z 307.791,A -85,B 0,C 180,E1 -13642.679,E2 -13642.679} C_VEL
LIN {X 0,Y 347.748,Z 307.788,A -85,B 0,C 180,E1 -13645.956,E2 -13645.956} C_VEL
LIN {X 0,Y 347.74,Z 307.785,A -85,B 0,C 180,E1 -13649.651,E2 -13649.651} C_VEL
LIN {X 0,Y 347.739,Z 307.783,A -85,B 0,C 180,E1 -13653.6,E2 -13653.6} C_VEL
LIN {X 0,Y 347.77,Z 307.791,A -85,B 0,C 180,E1 -13656.16,E2 -13656.16} C_VEL
LIN {X 0,Y 347.806,Z 307.783,A -85,B 0,C 180,E1 -13659.909,E2 -13659.909} C_VEL
LIN {X 0,Y 347.832,Z 307.767,A -85,B 0,C 180,E1 -13663.568,E2 -13663.568} C_VEL
LIN {X 0,Y 347.89,Z 307.766,A -85,B 0,C 180,E1 -13667.16,E2 -13667.16} C_VEL
LIN {X 0,Y 347.935,Z 307.771,A -85,B 0,C 180,E1 -13670.7,E2 -13670.7} C_VEL
LIN {X 0,Y 348.043,Z 307.738,A -85,B 0,C 180,E1 -13674.205,E2 -13674.205} C_VEL
LIN {X 0,Y 348.205,Z 307.734,A -85,B 0,C 180,E1 -13677.686,E2 -13677.686} C_VEL
LIN {X 0,Y 348.325,Z 307.702,A -85,B 0,C 180,E1 -13680,E2 -13680} C_VEL
LIN {X 0,Y 348.195,Z 307.738,A -85,B 0,C 180,E1 -13682.313,E2 -13682.313} C_VEL
LIN {X 0,Y 348.072,Z 307.746,A -85,B 0,C 180,E1 -13686.958,E2 -13686.958} C_VEL
LIN {X 0,Y 347.896,Z 307.756,A -85,B 0,C 180,E1 -13690.475,E2 -13690.475} C_VEL
LIN {X 0,Y 347.898,Z 307.774,A -85,B 0,C 180,E1 -13694.15,E2 -13694.15} C_VEL
LIN {X 0,Y 347.89,Z 307.772,A -85,B 0,C 180,E1 -13698.29,E2 -13698.29} C_VEL
LIN {X 0,Y 347.767,Z 307.775,A -85,B 0,C 180,E1 -13701.626,E2 -13701.626} C_VEL
LIN {X 0,Y 347.768,Z 307.787,A -85,B 0,C 180,E1 -13705.112,E2 -13705.112} C_VEL
LIN {X 0,Y 347.736,Z 307.788,A -85,B 0,C 180,E1 -13707.7,E2 -13707.7} C_VEL
LIN {X 0,Y 347.74,Z 307.796,A -85,B 0,C 180,E1 -13710.349,E2 -13710.349} C_VEL
LIN {X 0,Y 347.747,Z 307.793,A -85,B 0,C 180,E1 -13714.044,E2 -13714.044} C_VEL
LIN {X 0,Y 347.76,Z 307.793,A -85,B 0,C 180,E1 -13717.321,E2 -13717.321} C_VEL
LIN {X 0,Y 347.811,Z 307.99,A -85,B 0,C 180,E1 -13718.22,E2 -13718.22} C_VEL
LIN {X 0,Y 349.664,Z 315.991,A -85,B 0,C 180,E1 -13721.55,E2 -13721.55} C_VEL
LIN {X 0,Y 351.788,Z 324.99,A -85,B 0,C 180,E1 -13725.066,E2 -13725.066} C_VEL
LIN {X 0,Y 354.057,Z 334.474,A -85,B 0,C 180,E1 -13728.532,E2 -13728.532} C_VEL
LIN {X 0,Y 356.741,Z 345.613,A -85,B 0,C 180,E1 -13732.359,E2 -13732.359} C_VEL
LIN {X 0,Y 356.616,Z 347.882,A -85,B 0,C 180,E1 -13733.053,E2 -13733.053} C_VEL
LIN {X 0,Y 354.304,Z 359.338,A -85,B 0,C 180,E1 -13736.42,E2 -13736.42} C_VEL
LIN {X 0,Y 351.857,Z 373.668,A -85,B 0,C 180,E1 -13740.553,E2 -13740.553} C_VEL
LIN {X 0,Y 356.42,Z 398.635,A -85,B 0,C 180,E1 -13741.617,E2 -13741.617} C_VEL
LIN {X 0,Y 358.507,Z 414.283,A -85,B 0,C 180,E1 -13742.457,E2 -13742.457} C_VEL
LIN {X 0,Y 359.595,Z 427.19,A -85,B 0,C 180,E1 -13743.288,E2 -13743.288} C_VEL
LIN {X 0,Y 359.789,Z 433.999,A -85,B 0,C 180,E1 -13743.772,E2 -13743.772} C_VEL
LIN {X 0,Y 358.167,Z 447.137,A -85,B 0,C 180,E1 -13744.737,E2 -13744.737} C_VEL
LIN {X 0,Y 356.169,Z 460.854,A -85,B 0,C 180,E1 -13745.985,E2 -13745.985} C_VEL
LIN {X 0,Y 354.012,Z 474.535,A -85,B 0,C 180,E1 -13747.533,E2 -13747.533} C_VEL
LIN {X 0,Y 352.111,Z 487.014,A -85,B 0,C 180,E1 -13749.281,E2 -13749.281} C_VEL
LIN {X 0,Y 350.52,Z 497.233,A -85,B 0,C 180,E1 -13750.997,E2 -13750.997} C_VEL
LIN {X 0,Y 349.013,Z 507.279,A -85,B 0,C 180,E1 -13753.023,E2 -13753.023} C_VEL
LIN {X 0,Y 347.923,Z 515.69,A -85,B 0,C 180,E1 -13755.076,E2 -13755.076} C_VEL
LIN {X 0,Y 347.137,Z 522.667,A -85,B 0,C 180,E1 -13757.132,E2 -13757.132} C_VEL
LIN {X 0,Y 346.635,Z 529.155,A -85,B 0,C 180,E1 -13759.486,E2 -13759.486} C_VEL
LIN {X 0,Y 346.497,Z 534.187,A -85,B 0,C 180,E1 -13761.838,E2 -13761.838} C_VEL
LIN {X 0,Y 346.58,Z 537.883,A -85,B 0,C 180,E1 -13764.181,E2 -13764.181} C_VEL
LIN {X 0,Y 346.684,Z 540.321,A -85,B 0,C 180,E1 -13766.514,E2 -13766.514} C_VEL
LIN {X 0,Y 346.793,Z 541.551,A -85,B 0,C 180,E1 -13768.839,E2 -13768.839} C_VEL
LIN {X 0,Y 346.795,Z 541.55,A -85,B 0,C 180,E1 -13771.161,E2 -13771.161} C_VEL
LIN {X 0,Y 346.708,Z 540.32,A -85,B 0,C 180,E1 -13773.487,E2 -13773.487} C_VEL
LIN {X 0,Y 346.625,Z 537.879,A -85,B 0,C 180,E1 -13775.819,E2 -13775.819} C_VEL
LIN {X 0,Y 346.538,Z 534.169,A -85,B 0,C 180,E1 -13778.162,E2 -13778.162} C_VEL
LIN {X 0,Y 346.663,Z 529.127,A -85,B 0,C 180,E1 -13780.513,E2 -13780.513} C_VEL
LIN {X 0,Y 347.163,Z 522.638,A -85,B 0,C 180,E1 -13782.867,E2 -13782.867} C_VEL
LIN {X 0,Y 348.052,Z 514.509,A -85,B 0,C 180,E1 -13785.219,E2 -13785.219} C_VEL
LIN {X 0,Y 349.2,Z 505.854,A -85,B 0,C 180,E1 -13787.269,E2 -13787.269} C_VEL
LIN {X 0,Y 350.888,Z 495.465,A -85,B 0,C 180,E1 -13789.298,E2 -13789.298} C_VEL
LIN {X 0,Y 352.449,Z 484.826,A -85,B 0,C 180,E1 -13791.035,E2 -13791.035} C_VEL
LIN {X 0,Y 354.27,Z 473.27,A -85,B 0,C 180,E1 -13792.604,E2 -13792.604} C_VEL
LIN {X 0,Y 356.22,Z 460.723,A -85,B 0,C 180,E1 -13794.012,E2 -13794.012} C_VEL
LIN {X 0,Y 358.131,Z 446.989,A -85,B 0,C 180,E1 -13795.267,E2 -13795.267} C_VEL
LIN {X 0,Y 360.071,Z 433.601,A -85,B 0,C 180,E1 -13796.362,E2 -13796.362} C_VEL
LIN {X 0,Y 360.663,Z 418.438,A -85,B 0,C 180,E1 -13797.726,E2 -13797.726} C_VEL
LIN {X 0,Y 360.319,Z 405.134,A -85,B 0,C 180,E1 -13798.843,E2 -13798.843} C_VEL
LIN {X 0,Y 358.947,Z 393.635,A -85,B 0,C 180,E1 -13799.843,E2 -13799.843} C_VEL
LIN {X 0,Y 356.268,Z 380.404,A -85,B 0,C 180,E1 -13801.047,E2 -13801.047} C_VEL
LIN {X 0,Y 354.134,Z 371.547,A -85,B 0,C 180,E1 -13801.908,E2 -13801.908} C_VEL
LIN {X 0,Y 357.091,Z 361.236,A -85,B 0,C 180,E1 -13805.493,E2 -13805.493} C_VEL
LIN {X 0,Y 358.951,Z 356.296,A -85,B 0,C 180,E1 -13807.37,E2 -13807.37} C_VEL
LIN {X 0,Y 359.205,Z 355.057,A -85,B 0,C 180,E1 -13807.902,E2 -13807.902} C_VEL
LIN {X 0,Y 358.734,Z 352.092,A -85,B 0,C 180,E1 -13809.448,E2 -13809.448} C_VEL
LIN {X 0,Y 357.644,Z 348.116,A -85,B 0,C 180,E1 -13811.923,E2 -13811.923} C_VEL
LIN {X 0,Y 356.369,Z 343.942,A -85,B 0,C 180,E1 -13815.232,E2 -13815.232} C_VEL
LIN {X 0,Y 355.514,Z 341.563,A -85,B 0,C 180,E1 -13817.768,E2 -13817.768} C_VEL
LIN {X 0,Y 354.748,Z 339.597,A -85,B 0,C 180,E1 -13820.657,E2 -13820.657} C_VEL
LIN {X 0,Y 353.976,Z 338.446,A -85,B 0,C 180,E1 -13823.442,E2 -13823.442} C_VEL
LIN {X 0,Y 353.039,Z 337.892,A -85,B 0,C 180,E1 -13826.731,E2 -13826.731} C_VEL
LIN {X 0,Y 352.186,Z 338.004,A -85,B 0,C 180,E1 -13830.074,E2 -13830.074} C_VEL
LIN {X 0,Y 351.694,Z 338.656,A -85,B 0,C 180,E1 -13832.928,E2 -13832.928} C_VEL
LIN {X 0,Y 353.29,Z 341.579,A -85,B 0,C 180,E1 -13833.533,E2 -13833.533} C_VEL
LIN {X 0,Y 354.281,Z 342.673,A -85,B 0,C 180,E1 -13833.84,E2 -13833.84} C_VEL
LIN {X 0,Y 355.145,Z 344.506,A -85,B 0,C 180,E1 -13834.192,E2 -13834.192} C_VEL
LIN {X 0,Y 356.222,Z 345.807,A -85,B 0,C 180,E1 -13834.522,E2 -13834.522} C_VEL
LIN {X 0,Y 361.361,Z 355.673,A -85,B 0,C 180,E1 -13836.423,E2 -13836.423} C_VEL
LIN {X 0,Y 364.444,Z 363.394,A -85,B 0,C 180,E1 -13837.766,E2 -13837.766} C_VEL
LIN {X 0,Y 365.436,Z 366.423,A -85,B 0,C 180,E1 -13838.259,E2 -13838.259} C_VEL
LIN {X 0,Y 363.329,Z 379.159,A -85,B 0,C 180,E1 -13839.624,E2 -13839.624} C_VEL
LIN {X 0,Y 361.211,Z 389.82,A -85,B 0,C 180,E1 -13840.98,E2 -13840.98} C_VEL
LIN {X 0,Y 358.951,Z 400.344,A -85,B 0,C 180,E1 -13842.628,E2 -13842.628} C_VEL
LIN {X 0,Y 356.675,Z 410.36,A -85,B 0,C 180,E1 -13844.573,E2 -13844.573} C_VEL
LIN {X 0,Y 354.886,Z 417.382,A -85,B 0,C 180,E1 -13846.253,E2 -13846.253} C_VEL
LIN {X 0,Y 353.35,Z 423.116,A -85,B 0,C 180,E1 -13847.946,E2 -13847.946} C_VEL
LIN {X 0,Y 351.708,Z 429.092,A -85,B 0,C 180,E1 -13850.221,E2 -13850.221} C_VEL
LIN {X 0,Y 350.542,Z 432.425,A -85,B 0,C 180,E1 -13851.932,E2 -13851.932} C_VEL
LIN {X 0,Y 349.987,Z 434.112,A -85,B 0,C 180,E1 -13853.08,E2 -13853.08} C_VEL
LIN {X 0,Y 349.254,Z 436.208,A -85,B 0,C 180,E1 -13855.383,E2 -13855.383} C_VEL
LIN {X 0,Y 348.545,Z 436.844,A -85,B 0,C 180,E1 -13857.689,E2 -13857.689} C_VEL
LIN {X 0,Y 348.36,Z 436.564,A -85,B 0,C 180,E1 -13858.844,E2 -13858.844} C_VEL
LIN {X 0,Y 348.043,Z 435.886,A -85,B 0,C 180,E1 -13860,E2 -13860} C_VEL
LIN {X 0,Y 348.003,Z 434.787,A -85,B 0,C 180,E1 -13861.157,E2 -13861.157} C_VEL
LIN {X 0,Y 347.878,Z 433.317,A -85,B 0,C 180,E1 -13862.316,E2 -13862.316} C_VEL
LIN {X 0,Y 347.84,Z 430.305,A -85,B 0,C 180,E1 -13864.055,E2 -13864.055} C_VEL
LIN {X 0,Y 348.187,Z 426.278,A -85,B 0,C 180,E1 -13865.792,E2 -13865.792} C_VEL
LIN {X 0,Y 348.539,Z 421.2,A -85,B 0,C 180,E1 -13867.531,E2 -13867.531} C_VEL
LIN {X 0,Y 349.058,Z 413.788,A -85,B 0,C 180,E1 -13869.562,E2 -13869.562} C_VEL
LIN {X 0,Y 349.619,Z 405.89,A -85,B 0,C 180,E1 -13871.303,E2 -13871.303} C_VEL
LIN {X 0,Y 350.29,Z 396.313,A -85,B 0,C 180,E1 -13873.045,E2 -13873.045} C_VEL
LIN {X 0,Y 351.224,Z 385.682,A -85,B 0,C 180,E1 -13874.633,E2 -13874.633} C_VEL
LIN {X 0,Y 352.161,Z 373.867,A -85,B 0,C 180,E1 -13876.075,E2 -13876.075} C_VEL
LIN {X 0,Y 353.047,Z 360.856,A -85,B 0,C 180,E1 -13877.374,E2 -13877.374} C_VEL
LIN {X 0,Y 353.934,Z 347.076,A -85,B 0,C 180,E1 -13878.45,E2 -13878.45} C_VEL
LIN {X 0,Y 350.787,Z 333.905,A -85,B 0,C 180,E1 -13879.425,E2 -13879.425} C_VEL
LIN {X 0,Y 347.196,Z 319.752,A -85,B 0,C 180,E1 -13880.283,E2 -13880.283} C_VEL
LIN {X 0,Y 347.204,Z 315.363,A -85,B 0,C 180,E1 -13884.372,E2 -13884.372} C_VEL
LIN {X 0,Y 347.216,Z 311.87,A -85,B 0,C 180,E1 -13887.745,E2 -13887.745} C_VEL
LIN {X 0,Y 347.233,Z 309.176,A -85,B 0,C 180,E1 -13890.398,E2 -13890.398} C_VEL
LIN {X 0,Y 347.295,Z 307.852,A -85,B 0,C 180,E1 -13891.795,E2 -13891.795} C_VEL
LIN {X 0,Y 347.553,Z 307.812,A -85,B 0,C 180,E1 -13894.486,E2 -13894.486} C_VEL
LIN {X 0,Y 347.766,Z 307.79,A -85,B 0,C 180,E1 -13897.986,E2 -13897.986} C_VEL
LIN {X 0,Y 347.753,Z 307.788,A -85,B 0,C 180,E1 -13901.83,E2 -13901.83} C_VEL
LIN {X 0,Y 347.749,Z 307.973,A -85,B 0,C 180,E1 -13903.804,E2 -13903.804} C_VEL
LIN {X 0,Y 348.399,Z 311.509,A -85,B 0,C 180,E1 -13906.697,E2 -13906.697} C_VEL
LIN {X 0,Y 348.636,Z 313.552,A -85,B 0,C 180,E1 -13908.299,E2 -13908.299} C_VEL
LIN {X 0,Y 348.65,Z 317.426,A -85,B 0,C 180,E1 -13911.325,E2 -13911.325} C_VEL
LIN {X 0,Y 348.61,Z 321.238,A -85,B 0,C 180,E1 -13914.222,E2 -13914.222} C_VEL
LIN {X 0,Y 348.554,Z 326.318,A -85,B 0,C 180,E1 -13917.872,E2 -13917.872} C_VEL
LIN {X 0,Y 348.556,Z 329.854,A -85,B 0,C 180,E1 -13920.266,E2 -13920.266} C_VEL
LIN {X 0,Y 355.78,Z 347.133,A -85,B 0,C 180,E1 -13921.483,E2 -13921.483} C_VEL
LIN {X 0,Y 360.535,Z 360.577,A -85,B 0,C 180,E1 -13922.541,E2 -13922.541} C_VEL
LIN {X 0,Y 363.005,Z 368.953,A -85,B 0,C 180,E1 -13923.254,E2 -13923.254} C_VEL
LIN {X 0,Y 361.986,Z 382.815,A -85,B 0,C 180,E1 -13924.188,E2 -13924.188} C_VEL
LIN {X 0,Y 360.558,Z 395.373,A -85,B 0,C 180,E1 -13925.223,E2 -13925.223} C_VEL
LIN {X 0,Y 358.656,Z 409.148,A -85,B 0,C 180,E1 -13926.621,E2 -13926.621} C_VEL
LIN {X 0,Y 356.776,Z 421.553,A -85,B 0,C 180,E1 -13928.172,E2 -13928.172} C_VEL
LIN {X 0,Y 355.132,Z 431.93,A -85,B 0,C 180,E1 -13929.737,E2 -13929.737} C_VEL
LIN {X 0,Y 353.392,Z 441.532,A -85,B 0,C 180,E1 -13931.446,E2 -13931.446} C_VEL
LIN {X 0,Y 351.64,Z 450.909,A -85,B 0,C 180,E1 -13933.452,E2 -13933.452} C_VEL
LIN {X 0,Y 350.319,Z 458.695,A -85,B 0,C 180,E1 -13935.477,E2 -13935.477} C_VEL
LIN {X 0,Y 349.054,Z 465.935,A -85,B 0,C 180,E1 -13937.795,E2 -13937.795} C_VEL
LIN {X 0,Y 348.11,Z 471.668,A -85,B 0,C 180,E1 -13940.118,E2 -13940.118} C_VEL
LIN {X 0,Y 347.494,Z 475.845,A -85,B 0,C 180,E1 -13942.315,E2 -13942.315} C_VEL
LIN {X 0,Y 347.043,Z 478.496,A -85,B 0,C 180,E1 -13944.188,E2 -13944.188} C_VEL
LIN {X 0,Y 346.93,Z 480.749,A -85,B 0,C 180,E1 -13946.516,E2 -13946.516} C_VEL
LIN {X 0,Y 346.722,Z 481.907,A -85,B 0,C 180,E1 -13948.838,E2 -13948.838} C_VEL
LIN {X 0,Y 346.721,Z 481.919,A -85,B 0,C 180,E1 -13951.161,E2 -13951.161} C_VEL
LIN {X 0,Y 346.911,Z 480.814,A -85,B 0,C 180,E1 -13953.484,E2 -13953.484} C_VEL
LIN {X 0,Y 347.041,Z 478.614,A -85,B 0,C 180,E1 -13955.811,E2 -13955.811} C_VEL
LIN {X 0,Y 347.587,Z 475.23,A -85,B 0,C 180,E1 -13958.136,E2 -13958.136} C_VEL
LIN {X 0,Y 348.282,Z 470.595,A -85,B 0,C 180,E1 -13960.463,E2 -13960.463} C_VEL
LIN {X 0,Y 349.321,Z 464.565,A -85,B 0,C 180,E1 -13962.786,E2 -13962.786} C_VEL
LIN {X 0,Y 350.659,Z 456.969,A -85,B 0,C 180,E1 -13965.102,E2 -13965.102} C_VEL
LIN {X 0,Y 352.05,Z 448.863,A -85,B 0,C 180,E1 -13967.125,E2 -13967.125} C_VEL
LIN {X 0,Y 353.844,Z 439.06,A -85,B 0,C 180,E1 -13969.13,E2 -13969.13} C_VEL
LIN {X 0,Y 355.579,Z 429.037,A -85,B 0,C 180,E1 -13970.84,E2 -13970.84} C_VEL
LIN {X 0,Y 357.248,Z 418.239,A -85,B 0,C 180,E1 -13972.39,E2 -13972.39} C_VEL
LIN {X 0,Y 359.334,Z 404.957,A -85,B 0,C 180,E1 -13973.943,E2 -13973.943} C_VEL
LIN {X 0,Y 361.083,Z 391.775,A -85,B 0,C 180,E1 -13975.199,E2 -13975.199} C_VEL
LIN {X 0,Y 362.581,Z 377.364,A -85,B 0,C 180,E1 -13976.302,E2 -13976.302} C_VEL
LIN {X 0,Y 363.174,Z 369.563,A -85,B 0,C 180,E1 -13976.8,E2 -13976.8} C_VEL
LIN {X 0,Y 359.084,Z 356.091,A -85,B 0,C 180,E1 -13977.933,E2 -13977.933} C_VEL
LIN {X 0,Y 353.808,Z 342.011,A -85,B 0,C 180,E1 -13978.999,E2 -13978.999} C_VEL
LIN {X 0,Y 348.588,Z 329.88,A -85,B 0,C 180,E1 -13979.841,E2 -13979.841} C_VEL
LIN {X 0,Y 348.553,Z 327.767,A -85,B 0,C 180,E1 -13981.253,E2 -13981.253} C_VEL
LIN {X 0,Y 347.91,Z 326.54,A -85,B 0,C 180,E1 -13982.197,E2 -13982.197} C_VEL
LIN {X 0,Y 345.077,Z 324.994,A -85,B 0,C 180,E1 -13983.748,E2 -13983.748} C_VEL
LIN {X 0,Y 342.696,Z 323.798,A -85,B 0,C 180,E1 -13985.006,E2 -13985.006} C_VEL
LIN {X 0,Y 341.716,Z 322.738,A -85,B 0,C 180,E1 -13985.975,E2 -13985.975} C_VEL
LIN {X 0,Y 341.659,Z 322.309,A -85,B 0,C 180,E1 -13986.3,E2 -13986.3} C_VEL
LIN {X 0,Y 341.745,Z 317.985,A -85,B 0,C 180,E1 -13989.607,E2 -13989.607} C_VEL
LIN {X 0,Y 341.562,Z 314.023,A -85,B 0,C 180,E1 -13992.766,E2 -13992.766} C_VEL
LIN {X 0,Y 341.056,Z 310.643,A -85,B 0,C 180,E1 -13995.523,E2 -13995.523} C_VEL
LIN {X 0,Y 340.673,Z 308.677,A -85,B 0,C 180,E1 -13997.215,E2 -13997.215} C_VEL
LIN {X 0,Y 340.699,Z 308.669,A -85,B 0,C 180,E1 -14000.247,E2 -14000.247} C_VEL
LIN {X 0,Y 340.71,Z 308.665,A -85,B 0,C 180,E1 -14003.559,E2 -14003.559} C_VEL
LIN {X 0,Y 340.692,Z 308.665,A -85,B 0,C 180,E1 -14006.153,E2 -14006.153} C_VEL
LIN {X 0,Y 340.723,Z 308.658,A -85,B 0,C 180,E1 -14010.034,E2 -14010.034} C_VEL
LIN {X 0,Y 340.711,Z 308.663,A -85,B 0,C 180,E1 -14013.012,E2 -14013.012} C_VEL
LIN {X 0,Y 340.741,Z 308.667,A -85,B 0,C 180,E1 -14015.637,E2 -14015.637} C_VEL
LIN {X 0,Y 340.734,Z 308.661,A -85,B 0,C 180,E1 -14019.473,E2 -14019.473} C_VEL
LIN {X 0,Y 340.792,Z 308.651,A -85,B 0,C 180,E1 -14021.981,E2 -14021.981} C_VEL
LIN {X 0,Y 340.869,Z 308.651,A -85,B 0,C 180,E1 -14025.705,E2 -14025.705} C_VEL
LIN {X 0,Y 340.848,Z 308.64,A -85,B 0,C 180,E1 -14029.305,E2 -14029.305} C_VEL
LIN {X 0,Y 341.002,Z 308.621,A -85,B 0,C 180,E1 -14032.897,E2 -14032.897} C_VEL
LIN {X 0,Y 341.166,Z 308.611,A -85,B 0,C 180,E1 -14037.639,E2 -14037.639} C_VEL
LIN {X 0,Y 341.276,Z 308.579,A -85,B 0,C 180,E1 -14040,E2 -14040} C_VEL
LIN {X 0,Y 341.156,Z 308.615,A -85,B 0,C 180,E1 -14042.361,E2 -14042.361} C_VEL
LIN {X 0,Y 341.041,Z 308.623,A -85,B 0,C 180,E1 -14047.102,E2 -14047.102} C_VEL
LIN {X 0,Y 340.848,Z 308.632,A -85,B 0,C 180,E1 -14050.694,E2 -14050.694} C_VEL
LIN {X 0,Y 340.863,Z 308.65,A -85,B 0,C 180,E1 -14054.325,E2 -14054.325} C_VEL
LIN {X 0,Y 340.837,Z 308.652,A -85,B 0,C 180,E1 -14058.466,E2 -14058.466} C_VEL
LIN {X 0,Y 340.717,Z 308.653,A -85,B 0,C 180,E1 -14061.842,E2 -14061.842} C_VEL
LIN {X 0,Y 340.719,Z 308.659,A -85,B 0,C 180,E1 -14065.668,E2 -14065.668} C_VEL
LIN {X 0,Y 340.707,Z 308.67,A -85,B 0,C 180,E1 -14069.674,E2 -14069.674} C_VEL
